C09139=1214.216,61.843,-46.084,-178.985,5.599,148.680
C09140=1214.211,62.093,-46.102,-178.982,5.599,148.680
C09141=1214.206,62.341,-46.118,-178.980,5.600,148.679
C09142=1214.201,62.591,-46.136,-178.978,5.601,148.678
C09143=1214.197,62.841,-46.152,-178.975,5.601,148.678
C09144=1214.192,63.090,-46.169,-178.972,5.602,148.677
C09145=1214.186,63.339,-46.186,-178.970,5.603,148.676
C09146=1214.182,63.589,-46.203,-178.967,5.604,148.676
C09147=1214.177,63.838,-46.220,-178.965,5.604,148.675
C09148=1214.172,64.088,-46.237,-178.962,5.605,148.675
C09149=1214.167,64.337,-46.255,-178.960,5.605,148.674
C09150=1214.162,64.586,-46.271,-178.957,5.606,148.674
C09151=1214.157,64.836,-46.288,-178.954,5.608,148.673
C09152=1214.152,65.085,-46.305,-178.952,5.608,148.672
C09153=1214.147,65.335,-46.322,-178.949,5.609,148.672
C09154=1214.142,65.583,-46.339,-178.947,5.610,148.671
C09155=1214.137,65.833,-46.356,-178.944,5.610,148.670
C09156=1214.133,66.082,-46.373,-178.942,5.611,148.670
C09157=1214.128,66.332,-46.390,-178.939,5.611,148.669
C09158=1214.123,66.582,-46.407,-178.937,5.612,148.669
C09159=1214.118,66.831,-46.425,-178.934,5.613,148.668
C09160=1214.113,67.080,-46.441,-178.932,5.613,148.667
C09161=1214.108,67.329,-46.458,-178.928,5.615,148.667
C09162=1214.103,67.579,-46.475,-178.926,5.616,148.666
C09163=1214.098,67.828,-46.493,-178.924,5.616,148.666
C09164=1214.094,68.078,-46.510,-178.921,5.617,148.665
C09165=1214.088,68.327,-46.527,-178.919,5.618,148.665
C09166=1214.084,68.576,-46.544,-178.916,5.618,148.664
C09167=1214.079,68.825,-46.561,-178.914,5.619,148.663
C09168=1214.074,69.075,-46.579,-178.911,5.619,148.663
C09169=1214.069,69.324,-46.596,-178.909,5.620,148.662
C09170=1214.064,69.574,-46.613,-178.906,5.622,148.662
C09171=1214.060,69.823,-46.630,-178.903,5.622,148.661
C09172=1214.054,70.072,-46.648,-178.900,5.623,148.660
C09173=1214.049,70.322,-46.665,-178.898,5.624,148.660
C09174=1214.044,70.571,-46.681,-178.896,5.624,148.659
C09175=1214.040,70.820,-46.699,-178.893,5.625,148.658
C09176=1214.035,71.070,-46.716,-178.891,5.626,148.658
C09177=1214.030,71.319,-46.733,-178.888,5.626,148.657
C09178=1214.025,71.569,-46.751,-178.885,5.628,148.657
C09179=1214.020,71.818,-46.768,-178.882,5.628,148.656
C09180=1214.016,72.067,-46.786,-178.880,5.629,148.656
C09181=1214.010,72.316,-46.803,-178.878,5.630,148.655
C09182=1214.006,72.565,-46.820,-178.875,5.630,148.654
C09183=1214.000,72.815,-46.838,-178.872,5.631,148.654
C09184=1213.995,73.065,-46.855,-178.870,5.632,148.653
C09185=1213.991,73.314,-46.872,-178.868,5.632,148.653
C09186=1213.986,73.564,-46.889,-178.864,5.634,148.652
C09187=1213.981,73.813,-46.907,-178.862,5.635,148.651
C09188=1213.976,74.062,-46.925,-178.860,5.635,148.651
C09189=1213.971,74.311,-46.942,-178.857,5.636,148.650
C09190=1213.966,74.561,-46.959,-178.854,5.636,148.649
C09191=1213.961,74.810,-46.977,-178.852,5.637,148.649
C09192=1213.957,75.060,-46.994,-178.850,5.638,148.648
C09193=1213.952,75.309,-47.012,-178.846,5.639,148.648
C09194=1213.946,75.557,-47.030,-178.844,5.640,148.647
C09195=1213.941,75.807,-47.047,-178.842,5.641,148.647
C09196=1213.937,76.056,-47.064,-178.839,5.641,148.646
C09197=1213.932,76.306,-47.082,-178.837,5.642,148.646
C09198=1213.927,76.555,-47.099,-178.834,5.643,148.645
C09199=1213.922,76.805,-47.117,-178.831,5.644,148.644
C09200=1213.917,77.054,-47.134,-178.828,5.645,148.644
C09201=1213.913,77.303,-47.152,-178.826,5.646,148.643
C09202=1213.907,77.553,-47.169,-178.824,5.646,148.642
C09203=1213.902,77.802,-47.187,-178.821,5.647,148.642
C09204=1213.898,78.051,-47.205,-178.819,5.648,148.641
C09205=1213.893,78.301,-47.222,-178.816,5.649,148.641
C09206=1213.888,78.550,-47.240,-178.813,5.650,148.640
C09207=1213.883,78.799,-47.258,-178.811,5.651,148.640
C09208=1213.878,79.049,-47.275,-178.808,5.651,148.639
C09209=1213.873,79.298,-47.293,-178.806,5.652,148.638
C09210=1213.868,79.547,-47.311,-178.803,5.653,148.638
C09211=1213.864,79.797,-47.328,-178.801,5.654,148.637
C09212=1213.859,80.046,-47.346,-178.798,5.655,148.637
C09213=1213.854,80.295,-47.364,-178.795,5.655,148.636
C09214=1213.849,80.545,-47.381,-178.793,5.656,148.636
C09215=1213.844,80.794,-47.399,-178.790,5.657,148.635
C09216=1213.839,81.062,-47.418,-178.787,5.658,148.634
C09217=1213.833,81.331,-47.437,-178.784,5.659,148.634
C09218=1213.828,81.599,-47.457,-178.782,5.660,148.633
C09219=1213.823,81.867,-47.476,-178.779,5.661,148.633
C09220=1213.818,82.117,-47.494,-178.776,5.662,148.632
C09221=1213.813,82.366,-47.511,-178.774,5.662,148.631
C09222=1213.808,82.616,-47.529,-178.772,5.663,148.631
C09223=1213.804,82.864,-47.547,-178.769,5.664,148.630
C09224=1213.799,83.114,-47.565,-178.766,5.665,148.629
C09225=1213.794,83.363,-47.583,-178.764,5.666,148.629
C09226=1213.789,83.613,-47.600,-178.761,5.667,148.628
C09227=1213.784,83.862,-47.618,-178.759,5.667,148.628
C09228=1213.779,84.111,-47.636,-178.756,5.668,148.627
C09229=1213.775,84.361,-47.654,-178.754,5.669,148.627
C09230=1213.770,84.610,-47.672,-178.751,5.670,148.626
C09231=1213.765,84.859,-47.690,-178.748,5.671,148.626
C09232=1213.760,85.108,-47.708,-178.746,5.672,148.625
C09233=1213.755,85.358,-47.726,-178.743,5.672,148.624
C09234=1213.750,85.607,-47.743,-178.741,5.673,148.624
C09235=1213.745,85.857,-47.761,-178.738,5.675,148.623
C09236=1213.740,86.106,-47.779,-178.735,5.675,148.623
C09237=1213.735,86.355,-47.797,-178.733,5.676,148.622
C09238=1213.731,86.605,-47.816,-178.730,5.677,148.621
C09239=1213.726,86.854,-47.834,-178.727,5.678,148.621
C09240=1213.721,87.103,-47.852,-178.725,5.679,148.620
C09241=1213.716,87.352,-47.870,-178.723,5.680,148.620
C09242=1213.711,87.601,-47.888,-178.720,5.680,148.619
C09243=1213.706,87.851,-47.905,-178.718,5.681,148.619
C09244=1213.701,88.100,-47.923,-178.715,5.683,148.618
C09245=1213.697,88.350,-47.942,-178.712,5.683,148.617
C09246=1213.692,88.599,-47.960,-178.710,5.684,148.617
C09247=1213.687,88.848,-47.978,-178.707,5.685,148.616
C09248=1213.682,89.098,-47.996,-178.705,5.685,148.616
C09249=1213.677,89.347,-48.014,-178.702,5.687,148.615
C09250=1213.672,89.596,-48.032,-178.699,5.688,148.615
C09251=1213.667,89.846,-48.051,-178.697,5.688,148.614
C09252=1213.662,90.095,-48.069,-178.695,5.689,148.614
C09253=1213.658,90.344,-48.087,-178.691,5.691,148.613
C09254=1213.653,90.593,-48.105,-178.689,5.692,148.612
C09255=1213.648,90.842,-48.123,-178.687,5.692,148.612
C09256=1213.644,91.092,-48.142,-178.684,5.693,148.611
C09257=1213.638,91.341,-48.160,-178.681,5.695,148.611
C09258=1213.633,91.590,-48.178,-178.679,5.695,148.610
C09259=1213.628,91.840,-48.196,-178.676,5.696,148.609
C09260=1213.623,92.089,-48.214,-178.674,5.697,148.609
C09261=1213.619,92.339,-48.232,-178.671,5.698,148.608
C09262=1213.614,92.587,-48.251,-178.668,5.699,148.608
C09263=1213.610,92.836,-48.269,-178.666,5.700,148.607
C09264=1213.604,93.086,-48.288,-178.663,5.700,148.607
C09265=1213.600,93.336,-48.306,-178.661,5.701,148.606
C09266=1213.595,93.585,-48.324,-178.658,5.703,148.606
C09267=1213.590,93.833,-48.343,-178.655,5.703,148.605
C09268=1213.585,94.083,-48.361,-178.653,5.704,148.605
C09269=1213.580,94.333,-48.380,-178.651,5.705,148.604
C09270=1213.575,94.582,-48.398,-178.647,5.706,148.603
C09271=1213.570,94.831,-48.416,-178.645,5.707,148.603
C09272=1213.566,95.080,-48.434,-178.643,5.708,148.602
C09273=1213.561,95.330,-48.453,-178.640,5.709,148.602
C09274=1213.556,95.579,-48.471,-178.637,5.710,148.601
C09275=1213.551,95.828,-48.490,-178.635,5.711,148.600
C09276=1213.546,96.077,-48.508,-178.633,5.711,148.600
C09277=1213.541,96.327,-48.527,-178.629,5.713,148.599
C09278=1213.536,96.576,-48.545,-178.627,5.714,148.599
C09279=1213.532,96.825,-48.564,-178.625,5.714,148.598
C09280=1213.527,97.075,-48.582,-178.622,5.715,148.598
C09281=1213.522,97.324,-48.600,-178.619,5.717,148.597
C09282=1213.517,97.573,-48.619,-178.617,5.717,148.597
C09283=1213.513,97.823,-48.638,-178.615,5.718,148.596
C09284=1213.507,98.072,-48.656,-178.612,5.719,148.596
C09285=1213.502,98.321,-48.675,-178.609,5.720,148.595
C09286=1213.498,98.570,-48.693,-178.607,5.721,148.595
C09287=1213.494,98.819,-48.712,-178.604,5.722,148.594
C09288=1213.488,99.068,-48.730,-178.601,5.724,148.593
C09289=1213.483,99.318,-48.748,-178.599,5.724,148.593
C09290=1213.479,99.567,-48.767,-178.596,5.725,148.592
C09291=1213.473,99.816,-48.786,-178.594,5.726,148.592
C09292=1213.469,100.065,-48.805,-178.591,5.727,148.591
C09293=1213.464,100.315,-48.824,-178.589,5.728,148.591
C09294=1213.459,100.564,-48.842,-178.586,5.729,148.590
C09295=1213.455,100.814,-48.861,-178.583,5.730,148.589
C09296=1213.449,101.062,-48.880,-178.581,5.731,148.589
C09297=1213.445,101.312,-48.898,-178.578,5.732,148.588
C09298=1213.441,101.561,-48.917,-178.576,5.733,148.588
C09299=1213.435,101.810,-48.936,-178.573,5.734,148.587
C09300=1213.430,102.059,-48.954,-178.570,5.735,148.587
C09301=1213.425,102.309,-48.973,-178.568,5.736,148.586
C09302=1213.421,102.558,-48.992,-178.565,5.737,148.586
C09303=1213.416,102.808,-49.011,-178.563,5.738,148.585
C09304=1213.411,103.056,-49.030,-178.560,5.739,148.585
C09305=1213.406,103.306,-49.048,-178.557,5.740,148.584
C09306=1213.401,103.555,-49.067,-178.555,5.741,148.583
C09307=1213.396,103.804,-49.085,-178.552,5.741,148.583
C09308=1213.392,104.054,-49.105,-178.550,5.742,148.582
C09309=1213.387,104.302,-49.124,-178.547,5.744,148.582
C09310=1213.381,104.552,-49.142,-178.545,5.745,148.581
C09311=1213.377,104.801,-49.161,-178.542,5.745,148.581
C09312=1213.372,105.051,-49.180,-178.539,5.747,148.580
C09313=1213.368,105.300,-49.199,-178.537,5.748,148.580
C09314=1213.362,105.549,-49.218,-178.534,5.748,148.579
C09315=1213.358,105.799,-49.236,-178.532,5.750,148.579
C09316=1213.353,106.048,-49.256,-178.529,5.751,148.578
C09317=1213.348,106.296,-49.274,-178.527,5.752,148.578
C09318=1213.343,106.546,-49.293,-178.524,5.753,148.577
C09319=1213.338,106.795,-49.312,-178.522,5.754,148.577
C09320=1213.334,107.064,-49.333,-178.519,5.755,148.576
C09321=1213.328,107.332,-49.353,-178.516,5.756,148.575
C09322=1213.324,107.600,-49.374,-178.513,5.757,148.575
C09323=1213.318,107.869,-49.394,-178.510,5.758,148.574
C09324=1213.313,108.119,-49.413,-178.508,5.759,148.574
C09325=1213.308,108.367,-49.432,-178.505,5.760,148.573
C09326=1213.304,108.617,-49.452,-178.502,5.761,148.573
C09327=1213.298,108.866,-49.470,-178.500,5.762,148.572
C09328=1213.294,109.115,-49.489,-178.497,5.764,148.571
C09329=1213.289,109.364,-49.509,-178.495,5.764,148.571
C09330=1213.285,109.614,-49.528,-178.492,5.765,148.570
C09331=1213.279,109.862,-49.547,-178.489,5.767,148.570
C09332=1213.274,110.113,-49.566,-178.487,5.768,148.569
C09333=1213.270,110.361,-49.585,-178.485,5.768,148.569
C09334=1213.265,110.611,-49.604,-178.482,5.770,148.568
C09335=1213.260,110.859,-49.623,-178.479,5.771,148.568
C09336=1213.256,111.109,-49.643,-178.477,5.772,148.567
C09337=1213.250,111.358,-49.662,-178.474,5.773,148.567
C09338=1213.246,111.608,-49.680,-178.471,5.774,148.566
C09339=1213.241,111.856,-49.700,-178.469,5.775,148.566
C09340=1213.236,112.106,-49.719,-178.466,5.776,148.565
C09341=1213.231,112.355,-49.738,-178.464,5.777,148.565
C09342=1213.226,112.604,-49.758,-178.461,5.778,148.564
C09343=1213.222,112.854,-49.777,-178.459,5.779,148.564
C09344=1213.217,113.102,-49.796,-178.456,5.780,148.563
C09345=1213.212,113.352,-49.816,-178.453,5.782,148.562
C09346=1213.207,113.601,-49.835,-178.451,5.782,148.562
C09347=1213.202,113.850,-49.854,-178.449,5.783,148.561
C09348=1213.198,114.099,-49.873,-178.445,5.785,148.561
C09349=1213.193,114.348,-49.893,-178.443,5.786,148.560
C09350=1213.188,114.598,-49.912,-178.441,5.786,148.560
C09351=1213.184,114.847,-49.931,-178.438,5.788,148.559
C09352=1213.179,115.096,-49.951,-178.435,5.789,148.559
C09353=1213.173,115.345,-49.970,-178.433,5.790,148.558
C09354=1213.169,115.595,-49.990,-178.430,5.791,148.558
C09355=1213.164,115.843,-50.008,-178.428,5.792,148.557
C09356=1213.159,116.093,-50.028,-178.425,5.793,148.557
C09357=1213.155,116.342,-50.048,-178.423,5.794,148.556
C09358=1213.149,116.591,-50.067,-178.420,5.795,148.556
C09359=1213.145,116.841,-50.087,-178.417,5.797,148.555
C09360=1213.141,117.090,-50.106,-178.415,5.797,148.555
C09361=1213.135,117.339,-50.125,-178.412,5.799,148.554
C09362=1213.130,117.588,-50.145,-178.409,5.800,148.553
C09363=1213.125,117.837,-50.164,-178.407,5.801,148.553
C09364=1213.120,118.087,-50.184,-178.404,5.802,148.552
C09365=1213.116,118.336,-50.203,-178.402,5.803,148.552
C09366=1213.111,118.584,-50.223,-178.399,5.804,148.551
C09367=1213.107,118.834,-50.242,-178.397,5.805,148.551
C09368=1213.102,119.083,-50.262,-178.394,5.806,148.550
C09369=1213.097,119.332,-50.281,-178.391,5.808,148.550
C09370=1213.092,119.582,-50.301,-178.389,5.808,148.549
C09371=1213.087,119.831,-50.321,-178.387,5.809,148.549
C09372=1213.083,120.079,-50.340,-178.383,5.811,148.548
C09373=1213.078,120.329,-50.360,-178.381,5.812,148.548
C09374=1213.073,120.579,-50.379,-178.378,5.813,148.547
C09375=1213.068,120.827,-50.399,-178.376,5.814,148.547
C09376=1213.063,121.077,-50.418,-178.373,5.815,148.546
C09377=1213.059,121.326,-50.439,-178.371,5.817,148.546
C09378=1213.054,121.575,-50.458,-178.368,5.817,148.545
C09379=1213.049,121.824,-50.478,-178.365,5.819,148.545
C09380=1213.044,122.074,-50.497,-178.363,5.820,148.544
C09381=1213.039,122.323,-50.518,-178.360,5.821,148.544
C09382=1213.034,122.572,-50.537,-178.358,5.822,148.543
C09383=1213.029,122.821,-50.557,-178.355,5.823,148.543
C09384=1213.026,123.070,-50.576,-178.352,5.824,148.542
C09385=1213.021,123.319,-50.596,-178.350,5.825,148.542
C09386=1213.016,123.568,-50.615,-178.347,5.827,148.541
C09387=1213.011,123.817,-50.636,-178.345,5.828,148.541
C09388=1213.006,124.067,-50.655,-178.342,5.829,148.540
C09389=1213.002,124.316,-50.675,-178.340,5.830,148.540
C09390=1212.997,124.565,-50.695,-178.337,5.831,148.539
C09391=1212.992,124.814,-50.715,-178.334,5.832,148.539
C09392=1212.987,125.064,-50.734,-178.332,5.833,148.538
C09393=1212.983,125.313,-50.755,-178.329,5.835,148.538
C09394=1212.977,125.562,-50.774,-178.327,5.836,148.537
C09395=1212.973,125.811,-50.794,-178.324,5.837,148.537
C09396=1212.968,126.060,-50.814,-178.322,5.838,148.536
C09397=1212.963,126.310,-50.834,-178.319,5.839,148.536
C09398=1212.959,126.559,-50.854,-178.316,5.841,148.535
C09399=1212.953,126.808,-50.874,-178.314,5.841,148.535
C09400=1212.948,127.057,-50.894,-178.311,5.843,148.534
C09401=1212.944,127.306,-50.914,-178.308,5.844,148.533
C09402=1212.939,127.555,-50.934,-178.306,5.845,148.533
C09403=1212.935,127.805,-50.954,-178.304,5.846,148.533
C09404=1212.930,128.053,-50.974,-178.300,5.848,148.532
C09405=1212.925,128.303,-50.994,-178.298,5.849,148.532
C09406=1212.920,128.552,-51.014,-178.296,5.849,148.531
C09407=1212.916,128.801,-51.034,-178.293,5.851,148.531
C09408=1212.911,129.050,-51.054,-178.290,5.852,148.530
C09409=1212.906,129.299,-51.073,-178.288,5.854,148.530
C09410=1212.901,129.548,-51.094,-178.285,5.854,148.529
C09411=1212.896,129.797,-51.115,-178.282,5.856,148.529
C09412=1212.891,130.047,-51.134,-178.280,5.857,148.528
C09413=1212.887,130.296,-51.155,-178.277,5.858,148.528
C09414=1212.882,130.545,-51.174,-178.275,5.859,148.527
C09415=1212.878,130.794,-51.195,-178.272,5.861,148.527
C09416=1212.872,131.043,-51.214,-178.270,5.862,148.526
C09417=1212.867,131.292,-51.235,-178.267,5.863,148.526
C09418=1212.863,131.541,-51.255,-178.264,5.864,148.525
C09419=1212.858,131.791,-51.275,-178.262,5.865,148.525
C09420=1212.854,132.040,-51.295,-178.259,5.867,148.524
C09421=1212.849,132.289,-51.316,-178.257,5.868,148.524
C09422=1212.844,132.539,-51.336,-178.254,5.869,148.523
C09423=1212.839,132.788,-51.356,-178.252,5.870,148.523
C09424=1212.834,133.056,-51.378,-178.249,5.871,148.522
C09425=1212.829,133.325,-51.400,-178.246,5.873,148.522
C09426=1212.823,133.594,-51.422,-178.243,5.874,148.521
C09427=1212.819,133.862,-51.443,-178.241,5.876,148.521
C09428=1212.814,134.111,-51.464,-178.237,5.877,148.520
C09429=1212.809,134.360,-51.484,-178.235,5.878,148.520
C09430=1212.804,134.609,-51.504,-178.232,5.879,148.519
C09431=1212.800,134.858,-51.525,-178.230,5.880,148.519
C09432=1212.795,135.108,-51.546,-178.227,5.882,148.518
C09433=1212.790,135.357,-51.565,-178.225,5.883,148.518
C09434=1212.786,135.606,-51.586,-178.222,5.885,148.517
C09435=1212.781,135.855,-51.606,-178.220,5.885,148.517
C09436=1212.775,136.104,-51.627,-178.217,5.887,148.516
C09437=1212.771,136.353,-51.647,-178.215,5.888,148.516
C09438=1212.767,136.602,-51.667,-178.212,5.889,148.515
C09439=1212.761,136.851,-51.688,-178.209,5.890,148.515
C09440=1212.757,137.100,-51.708,-178.206,5.892,148.514
C09441=1212.752,137.349,-51.728,-178.204,5.893,148.514
C09442=1212.747,137.599,-51.749,-178.201,5.895,148.513
C09443=1212.743,137.848,-51.770,-178.199,5.895,148.513
C09444=1212.738,138.096,-51.790,-178.196,5.897,148.512
C09445=1212.733,138.346,-51.811,-178.194,5.898,148.512
C09446=1212.729,138.595,-51.832,-178.191,5.899,148.511
C09447=1212.724,138.844,-51.851,-178.189,5.900,148.511
C09448=1212.719,139.094,-51.872,-178.186,5.902,148.510
C09449=1212.714,139.342,-51.893,-178.184,5.903,148.510
C09450=1212.709,139.592,-51.913,-178.180,5.904,148.509
C09451=1212.705,139.841,-51.934,-178.178,5.905,148.509
C09452=1212.700,140.090,-51.954,-178.176,5.907,148.509
C09453=1212.695,140.339,-51.975,-178.173,5.908,148.508
C09454=1212.691,140.588,-51.996,-178.170,5.909,148.508
C09455=1212.685,140.837,-52.017,-178.168,5.910,148.507
C09456=1212.681,141.086,-52.037,-178.165,5.912,148.507
C09457=1212.676,141.335,-52.057,-178.163,5.913,148.506
C09458=1212.671,141.584,-52.078,-178.160,5.914,148.506
C09459=1212.667,141.833,-52.099,-178.158,5.915,148.505
C09460=1212.662,142.083,-52.120,-178.155,5.917,148.505
C09461=1212.658,142.332,-52.140,-178.152,5.918,148.504
C09462=1212.653,142.581,-52.161,-178.150,5.919,148.504
C09463=1212.649,142.830,-52.182,-178.147,5.921,148.503
C09464=1212.643,143.079,-52.203,-178.144,5.922,148.503
C09465=1212.639,143.328,-52.224,-178.142,5.924,148.502
C09466=1212.634,143.577,-52.245,-178.140,5.925,148.502
C09467=1212.629,143.826,-52.265,-178.136,5.926,148.501
C09468=1212.624,144.075,-52.286,-178.134,5.927,148.501
C09469=1212.620,144.324,-52.306,-178.132,5.929,148.501
C09470=1212.615,144.574,-52.327,-178.129,5.930,148.500
C09471=1212.610,144.822,-52.348,-178.126,5.931,148.500
C09472=1212.605,145.071,-52.369,-178.124,5.933,148.499
C09473=1212.601,145.321,-52.390,-178.121,5.934,148.499
C09474=1212.596,145.570,-52.411,-178.118,5.936,148.498
C09475=1212.592,145.819,-52.431,-178.116,5.936,148.498
C09476=1212.587,146.068,-52.452,-178.113,5.938,148.497
C09477=1212.582,146.317,-52.474,-178.111,5.939,148.497
C09478=1212.577,146.566,-52.495,-178.108,5.940,148.496
C09479=1212.572,146.815,-52.515,-178.106,5.941,148.496
C09480=1212.568,147.064,-52.536,-178.103,5.943,148.495
C09481=1212.563,147.313,-52.558,-178.100,5.945,148.495
C09482=1212.558,147.563,-52.579,-178.098,5.946,148.494
C09483=1212.554,147.812,-52.599,-178.095,5.947,148.494
C09484=1212.549,148.061,-52.620,-178.093,5.948,148.493
C09485=1212.545,148.309,-52.641,-178.090,5.950,148.493
C09486=1212.539,148.558,-52.662,-178.088,5.951,148.493
C09487=1212.535,148.808,-52.684,-178.085,5.952,148.492
C09488=1212.531,149.057,-52.705,-178.082,5.954,148.492
C09489=1212.525,149.306,-52.726,-178.080,5.955,148.491
C09490=1212.520,149.555,-52.747,-178.077,5.957,148.491
C09491=1212.516,149.804,-52.768,-178.075,5.957,148.490
C09492=1212.511,150.053,-52.789,-178.072,5.959,148.490
C09493=1212.506,150.303,-52.810,-178.069,5.961,148.490
C09494=1212.502,150.551,-52.831,-178.067,5.962,148.489
C09495=1212.497,150.800,-52.852,-178.064,5.963,148.489
C09496=1212.492,151.049,-52.874,-178.062,5.964,148.488
C09497=1212.487,151.298,-52.895,-178.059,5.966,148.488
C09498=1212.484,151.547,-52.916,-178.057,5.967,148.487
C09499=1212.478,151.797,-52.937,-178.054,5.969,148.487
C09500=1212.473,152.046,-52.958,-178.051,5.970,148.486
C09501=1212.469,152.294,-52.979,-178.049,5.971,148.486
C09502=1212.464,152.544,-53.000,-178.046,5.973,148.485
C09503=1212.460,152.793,-53.022,-178.044,5.974,148.485
C09504=1212.454,153.042,-53.043,-178.041,5.975,148.484
C09505=1212.450,153.291,-53.065,-178.038,5.977,148.484
C09506=1212.445,153.540,-53.085,-178.036,5.978,148.484
C09507=1212.441,153.789,-53.107,-178.033,5.980,148.483
C09508=1212.436,154.038,-53.128,-178.030,5.981,148.483
C09509=1212.431,154.287,-53.150,-178.028,5.982,148.482
C09510=1212.426,154.536,-53.170,-178.025,5.984,148.482
C09511=1212.422,154.785,-53.192,-178.023,5.985,148.481
C09512=1212.417,155.034,-53.214,-178.020,5.987,148.481
C09513=1212.412,155.283,-53.235,-178.017,5.988,148.481
C09514=1212.408,155.532,-53.257,-178.015,5.989,148.480
C09515=1212.403,155.782,-53.278,-178.012,5.991,148.480
C09516=1212.398,156.030,-53.299,-178.010,5.992,148.479
C09517=1212.393,156.279,-53.320,-178.007,5.993,148.479
C09518=1212.389,156.529,-53.342,-178.004,5.995,148.478
C09519=1212.384,156.777,-53.364,-178.002,5.996,148.478
C09520=1212.379,157.027,-53.385,-177.999,5.998,148.477
C09521=1212.375,157.276,-53.407,-177.996,5.999,148.477
C09522=1212.370,157.524,-53.428,-177.994,6.000,148.476
C09523=1212.365,157.774,-53.449,-177.992,6.002,148.476
C09524=1212.361,158.023,-53.471,-177.989,6.004,148.476
C09525=1212.356,158.271,-53.493,-177.986,6.005,148.475
C09526=1212.351,158.521,-53.514,-177.984,6.006,148.475
C09527=1212.347,158.770,-53.536,-177.982,6.007,148.474
C09528=1212.342,159.039,-53.560,-177.978,6.009,148.474
C09529=1212.337,159.308,-53.582,-177.976,6.011,148.473
C09530=1212.331,159.577,-53.606,-177.973,6.012,148.473
C09531=1212.327,159.846,-53.629,-177.970,6.014,148.472
C09532=1212.322,160.095,-53.650,-177.967,6.016,148.472
C09533=1212.317,160.344,-53.672,-177.965,6.017,148.472
C09534=1212.313,160.593,-53.694,-177.962,6.018,148.471
C09535=1212.308,160.841,-53.716,-177.959,6.020,148.471
C09536=1212.303,161.091,-53.737,-177.957,6.021,148.470
C09537=1212.298,161.340,-53.759,-177.955,6.023,148.470
C09538=1212.294,161.589,-53.780,-177.952,6.023,148.469
C09539=1212.289,161.838,-53.802,-177.949,6.025,148.469
C09540=1212.284,162.087,-53.824,-177.947,6.027,148.469
C09541=1212.280,162.335,-53.846,-177.945,6.028,148.468
C09542=1212.275,162.585,-53.868,-177.941,6.029,148.468
C09543=1212.270,162.834,-53.889,-177.939,6.031,148.467
C09544=1212.266,163.083,-53.911,-177.937,6.032,148.467
C09545=1212.261,163.332,-53.932,-177.934,6.034,148.466
C09546=1212.256,163.581,-53.954,-177.931,6.036,148.466
C09547=1212.252,163.830,-53.976,-177.929,6.037,148.465
C09548=1212.246,164.079,-53.999,-177.926,6.038,148.465
C09549=1212.242,164.328,-54.021,-177.923,6.040,148.465
C09550=1212.237,164.577,-54.042,-177.920,6.042,148.464
C09551=1212.233,164.826,-54.064,-177.918,6.043,148.464
C09552=1212.228,165.075,-54.086,-177.915,6.044,148.463
C09553=1212.224,165.324,-54.108,-177.913,6.046,148.463
C09554=1212.219,165.573,-54.130,-177.911,6.047,148.463
C09555=1212.214,165.822,-54.152,-177.908,6.049,148.462
C09556=1212.210,166.071,-54.173,-177.905,6.050,148.462
C09557=1212.205,166.319,-54.195,-177.903,6.051,148.461
C09558=1212.200,166.569,-54.217,-177.900,6.053,148.461
C09559=1212.195,166.818,-54.239,-177.897,6.055,148.460
C09560=1212.191,167.067,-54.261,-177.895,6.056,148.460
C09561=1212.186,167.316,-54.283,-177.892,6.058,148.460
C09562=1212.181,167.565,-54.305,-177.890,6.059,148.459
C09563=1212.177,167.814,-54.327,-177.887,6.060,148.459
C09564=1212.172,168.063,-54.349,-177.884,6.062,148.458
C09565=1212.167,168.312,-54.371,-177.882,6.064,148.458
C09566=1212.163,168.561,-54.394,-177.879,6.065,148.458
C09567=1212.158,168.809,-54.416,-177.877,6.066,148.457
C09568=1212.154,169.059,-54.438,-177.874,6.068,148.457
C09569=1212.149,169.307,-54.459,-177.871,6.070,148.456
C09570=1212.144,169.557,-54.482,-177.869,6.071,148.456
C09571=1212.139,169.806,-54.504,-177.866,6.072,148.455
C09572=1212.135,170.054,-54.526,-177.864,6.074,148.455
C09573=1212.131,170.304,-54.549,-177.861,6.076,148.455
C09574=1212.125,170.553,-54.571,-177.858,6.077,148.454
C09575=1212.121,170.802,-54.593,-177.856,6.079,148.454
C09576=1212.116,171.051,-54.615,-177.853,6.080,148.453
C09577=1212.112,171.299,-54.637,-177.851,6.081,148.453
C09578=1212.106,171.548,-54.660,-177.848,6.083,148.453
C09579=1212.102,171.798,-54.682,-177.846,6.085,148.452
C09580=1212.097,172.046,-54.703,-177.842,6.086,148.452
C09581=1212.093,172.295,-54.727,-177.840,6.087,148.451
C09582=1212.088,172.545,-54.749,-177.838,6.089,148.451
C09583=1212.083,172.793,-54.770,-177.835,6.091,148.451
C09584=1212.079,173.043,-54.792,-177.832,6.093,148.450
C09585=1212.074,173.291,-54.815,-177.830,6.094,148.450
C09586=1212.070,173.540,-54.837,-177.827,6.095,148.449
C09587=1212.065,173.790,-54.860,-177.824,6.097,148.449
C09588=1212.060,174.038,-54.883,-177.822,6.099,148.449
C09589=1212.056,174.287,-54.905,-177.820,6.100,148.448
C09590=1212.051,174.535,-54.927,-177.817,6.102,148.448
C09591=1212.046,174.785,-54.950,-177.814,6.103,148.447
C09592=1212.042,175.034,-54.972,-177.811,6.105,148.447
C09593=1212.037,175.283,-54.995,-177.809,6.106,148.446
C09594=1212.032,175.532,-55.017,-177.806,6.108,148.446
C09595=1212.028,175.780,-55.039,-177.804,6.110,148.446
C09596=1212.023,176.030,-55.062,-177.801,6.112,148.445
C09597=1212.018,176.279,-55.084,-177.799,6.113,148.445
C09598=1212.013,176.527,-55.107,-177.796,6.114,148.444
C09599=1212.009,176.777,-55.129,-177.793,6.116,148.444
C09600=1212.005,177.025,-55.152,-177.791,6.118,148.444
C09601=1211.999,177.274,-55.174,-177.789,6.119,148.443
C09602=1211.995,177.523,-55.197,-177.786,6.120,148.443
C09603=1211.990,177.773,-55.219,-177.783,6.122,148.443
C09604=1211.986,178.021,-55.242,-177.781,6.124,148.442
C09605=1211.981,178.270,-55.264,-177.778,6.125,148.442
C09606=1211.977,178.519,-55.287,-177.775,6.127,148.441
C09607=1211.971,178.768,-55.309,-177.773,6.128,148.441
C09608=1211.967,179.017,-55.332,-177.770,6.130,148.441
C09609=1211.963,179.266,-55.356,-177.768,6.131,148.440
C09610=1211.958,179.515,-55.378,-177.765,6.133,148.440
C09611=1211.953,179.763,-55.401,-177.763,6.135,148.439
C09612=1211.949,180.013,-55.423,-177.759,6.136,148.439
C09613=1211.944,180.262,-55.446,-177.757,6.138,148.439
C09614=1211.939,180.510,-55.468,-177.755,6.139,148.438
C09615=1211.934,180.760,-55.491,-177.752,6.141,148.438
C09616=1211.930,181.008,-55.514,-177.749,6.143,148.437
C09617=1211.925,181.258,-55.536,-177.747,6.145,148.437
C09618=1211.921,181.506,-55.559,-177.744,6.146,148.437
C09619=1211.916,181.755,-55.582,-177.742,6.147,148.436
C09620=1211.912,182.004,-55.604,-177.739,6.149,148.436
C09621=1211.907,182.253,-55.628,-177.736,6.151,148.435
C09622=1211.902,182.502,-55.651,-177.734,6.153,148.435
C09623=1211.898,182.750,-55.673,-177.731,6.154,148.435
C09624=1211.893,183.000,-55.696,-177.729,6.155,148.434
C09625=1211.889,183.249,-55.719,-177.726,6.157,148.434
C09626=1211.884,183.497,-55.742,-177.723,6.159,148.434
C09627=1211.879,183.746,-55.765,-177.721,6.161,148.433
C09628=1211.875,183.995,-55.787,-177.718,6.163,148.433
C09629=1211.870,184.245,-55.810,-177.716,6.164,148.432
C09630=1211.866,184.493,-55.833,-177.713,6.165,148.432
C09631=1211.861,184.742,-55.856,-177.710,6.167,148.432
C09632=1211.855,185.011,-55.881,-177.708,6.169,148.431
C09633=1211.851,185.281,-55.906,-177.705,6.171,148.431
C09634=1211.846,185.551,-55.931,-177.702,6.172,148.431
C09635=1211.840,185.820,-55.956,-177.699,6.174,148.430
C09636=1211.836,186.069,-55.979,-177.697,6.176,148.430
C09637=1211.832,186.318,-56.002,-177.694,6.178,148.429
C09638=1211.827,186.567,-56.025,-177.691,6.179,148.429
C09639=1211.823,186.816,-56.047,-177.689,6.180,148.428
C09640=1211.818,187.065,-56.071,-177.686,6.182,148.428
C09641=1211.813,187.314,-56.094,-177.684,6.184,148.428
C09642=1211.808,187.563,-56.117,-177.681,6.186,148.427
C09643=1211.804,187.812,-56.140,-177.679,6.188,148.427
C09644=1211.799,188.061,-56.163,-177.675,6.189,148.427
C09645=1211.795,188.310,-56.187,-177.673,6.190,148.426
C09646=1211.790,188.559,-56.210,-177.671,6.192,148.426
C09647=1211.786,188.807,-56.233,-177.668,6.194,148.425
C09648=1211.781,189.056,-56.256,-177.665,6.196,148.425
C09649=1211.776,189.305,-56.279,-177.663,6.197,148.425
C09650=1211.771,189.554,-56.302,-177.660,6.199,148.424
C09651=1211.767,189.802,-56.325,-177.658,6.200,148.424
C09652=1211.763,190.052,-56.348,-177.655,6.202,148.424
C09653=1211.758,190.301,-56.372,-177.653,6.204,148.423
C09654=1211.753,190.550,-56.395,-177.650,6.206,148.423
C09655=1211.748,190.799,-56.419,-177.647,6.208,148.423
C09656=1211.744,191.047,-56.441,-177.645,6.209,148.422
C09657=1211.740,191.296,-56.465,-177.642,6.211,148.422
C09658=1211.734,191.545,-56.488,-177.640,6.212,148.422
C09659=1211.730,191.794,-56.511,-177.637,6.214,148.421
C09660=1211.725,192.042,-56.535,-177.634,6.216,148.421
C09661=1211.721,192.291,-56.558,-177.631,6.217,148.420
C09662=1211.716,192.540,-56.582,-177.629,6.219,148.420
C09663=1211.711,192.789,-56.605,-177.626,6.221,148.420
C09664=1211.707,193.038,-56.628,-177.624,6.223,148.419
C09665=1211.703,193.287,-56.651,-177.621,6.224,148.419
C09666=1211.698,193.536,-56.675,-177.619,6.226,148.418
C09667=1211.694,193.784,-56.699,-177.616,6.227,148.418
C09668=1211.689,194.033,-56.722,-177.613,6.229,148.418
C09669=1211.684,194.283,-56.745,-177.611,6.231,148.417
C09670=1211.679,194.532,-56.769,-177.608,6.233,148.417
C09671=1211.675,194.781,-56.792,-177.606,6.235,148.417
C09672=1211.670,195.029,-56.816,-177.603,6.237,148.416
C09673=1211.666,195.278,-56.840,-177.601,6.238,148.416
C09674=1211.661,195.527,-56.863,-177.598,6.239,148.416
C09675=1211.656,195.776,-56.886,-177.596,6.241,148.415
C09676=1211.652,196.024,-56.910,-177.593,6.243,148.415
C09677=1211.647,196.274,-56.934,-177.590,6.245,148.415
C09678=1211.642,196.523,-56.957,-177.588,6.247,148.414
C09679=1211.638,196.771,-56.981,-177.585,6.249,148.414
C09680=1211.633,197.020,-57.005,-177.582,6.250,148.414
C09681=1211.629,197.269,-57.028,-177.580,6.252,148.413
C09682=1211.624,197.517,-57.052,-177.578,6.253,148.413
C09683=1211.620,197.766,-57.075,-177.575,6.255,148.413
C09684=1211.615,198.016,-57.099,-177.572,6.257,148.412
C09685=1211.610,198.264,-57.123,-177.570,6.259,148.412
C09686=1211.606,198.513,-57.146,-177.567,6.261,148.412
C09687=1211.601,198.761,-57.170,-177.564,6.262,148.411
C09688=1211.597,199.010,-57.194,-177.562,6.264,148.411
C09689=1211.592,199.259,-57.217,-177.559,6.266,148.410
C09690=1211.588,199.508,-57.241,-177.556,6.268,148.410
C09691=1211.583,199.757,-57.264,-177.554,6.270,148.410
C09692=1211.578,200.005,-57.288,-177.551,6.272,148.409
C09693=1211.574,200.254,-57.312,-177.549,6.273,148.409
C09694=1211.569,200.503,-57.336,-177.546,6.274,148.409
C09695=1211.565,200.752,-57.359,-177.544,6.276,148.408
C09696=1211.560,201.001,-57.384,-177.541,6.278,148.408
C09697=1211.555,201.250,-57.408,-177.538,6.280,148.408
C09698=1211.551,201.499,-57.432,-177.536,6.282,148.407
C09699=1211.546,201.748,-57.455,-177.533,6.284,148.407
C09700=1211.542,201.996,-57.479,-177.530,6.285,148.407
C09701=1211.537,202.245,-57.502,-177.528,6.287,148.406
C09702=1211.533,202.494,-57.527,-177.525,6.289,148.406
C09703=1211.527,202.743,-57.551,-177.523,6.291,148.406
C09704=1211.523,202.991,-57.575,-177.520,6.293,148.405
C09705=1211.519,203.240,-57.599,-177.517,6.295,148.405
C09706=1211.515,203.489,-57.622,-177.515,6.296,148.405
C09707=1211.510,203.738,-57.646,-177.513,6.297,148.404
C09708=1211.506,203.986,-57.671,-177.510,6.299,148.404
C09709=1211.500,204.236,-57.694,-177.507,6.301,148.404
C09710=1211.496,204.484,-57.719,-177.505,6.303,148.403
C09711=1211.491,204.733,-57.742,-177.502,6.305,148.403
C09712=1211.487,204.982,-57.766,-177.499,6.307,148.403
C09713=1211.482,205.231,-57.791,-177.497,6.308,148.402
C09714=1211.478,205.479,-57.815,-177.494,6.310,148.402
C09715=1211.473,205.728,-57.838,-177.491,6.312,148.402
C09716=1211.469,205.977,-57.863,-177.489,6.314,148.401
C09717=1211.464,206.226,-57.888,-177.486,6.316,148.401
C09718=1211.460,206.475,-57.911,-177.483,6.318,148.401
C09719=1211.455,206.724,-57.935,-177.481,6.319,148.400
C09720=1211.451,206.972,-57.959,-177.478,6.321,148.400
C09721=1211.446,207.221,-57.984,-177.475,6.323,148.400
C09722=1211.441,207.470,-58.007,-177.473,6.325,148.399
C09723=1211.437,207.719,-58.032,-177.471,6.327,148.399
C09724=1211.432,207.968,-58.056,-177.468,6.329,148.399
C09725=1211.428,208.216,-58.080,-177.465,6.331,148.398
C09726=1211.423,208.464,-58.104,-177.463,6.333,148.398
C09727=1211.419,208.714,-58.129,-177.460,6.334,148.398
C09728=1211.414,208.963,-58.153,-177.458,6.335,148.397
C09729=1211.410,209.211,-58.177,-177.455,6.337,148.397
C09730=1211.404,209.460,-58.201,-177.453,6.339,148.397
C09731=1211.401,209.709,-58.226,-177.450,6.341,148.396
C09732=1211.396,209.958,-58.251,-177.447,6.343,148.396
C09733=1211.391,210.206,-58.275,-177.445,6.345,148.396
C09734=1211.387,210.455,-58.299,-177.442,6.346,148.395
C09735=1211.382,210.704,-58.324,-177.440,6.348,148.395
C09736=1211.377,210.975,-58.350,-177.436,6.351,148.395
C09737=1211.372,211.245,-58.376,-177.434,6.353,148.394
C09738=1211.367,211.515,-58.403,-177.431,6.355,148.394
C09739=1211.362,211.785,-58.429,-177.428,6.356,148.394
C09740=1211.358,212.034,-58.454,-177.426,6.358,148.393
C09741=1211.353,212.283,-58.478,-177.423,6.360,148.393
C09742=1211.349,212.531,-58.503,-177.421,6.362,148.393
C09743=1211.344,212.781,-58.528,-177.418,6.364,148.392
C09744=1211.340,213.029,-58.552,-177.415,6.366,148.392
C09745=1211.335,213.278,-58.576,-177.413,6.368,148.392
C09746=1211.331,213.527,-58.601,-177.410,6.370,148.392
C09747=1211.326,213.776,-58.625,-177.408,6.372,148.391
C09748=1211.321,214.024,-58.649,-177.405,6.373,148.391
C09749=1211.317,214.274,-58.675,-177.403,6.375,148.391
C09750=1211.312,214.522,-58.699,-177.400,6.377,148.390
C09751=1211.307,214.771,-58.723,-177.397,6.379,148.390
C09752=1211.304,215.020,-58.748,-177.395,6.381,148.390
C09753=1211.298,215.269,-58.772,-177.392,6.383,148.389
C09754=1211.294,215.516,-58.797,-177.389,6.384,148.389
C09755=1211.290,215.766,-58.822,-177.387,6.386,148.389
C09756=1211.285,216.014,-58.846,-177.385,6.388,148.388
C09757=1211.280,216.263,-58.871,-177.381,6.391,148.388
C09758=1211.276,216.512,-58.896,-177.379,6.393,148.388
C09759=1211.271,216.761,-58.920,-177.376,6.395,148.387
C09760=1211.266,217.009,-58.945,-177.373,6.397,148.387
C09761=1211.263,217.258,-58.970,-177.371,6.398,148.387
C09762=1211.258,217.507,-58.995,-177.368,6.400,148.387
C09763=1211.253,217.756,-59.020,-177.365,6.402,148.386
C09764=1211.249,218.004,-59.044,-177.363,6.404,148.386
C09765=1211.244,218.253,-59.069,-177.361,6.406,148.386
C09766=1211.240,218.502,-59.093,-177.358,6.408,148.385
C09767=1211.235,218.750,-59.118,-177.355,6.410,148.385
C09768=1211.231,218.999,-59.144,-177.353,6.412,148.385
C09769=1211.226,219.248,-59.168,-177.350,6.414,148.384
C09770=1211.222,219.497,-59.193,-177.348,6.415,148.384
C09771=1211.217,219.745,-59.218,-177.345,6.417,148.384
C09772=1211.213,219.994,-59.242,-177.343,6.419,148.384
C09773=1211.208,220.243,-59.267,-177.340,6.421,148.383
C09774=1211.203,220.491,-59.293,-177.337,6.423,148.383
C09775=1211.199,220.740,-59.317,-177.335,6.425,148.383
C09776=1211.194,220.989,-59.342,-177.332,6.427,148.382
C09777=1211.190,221.238,-59.368,-177.330,6.429,148.382
C09778=1211.185,221.487,-59.392,-177.327,6.430,148.382
C09779=1211.181,221.735,-59.418,-177.325,6.433,148.382
C09780=1211.176,221.984,-59.442,-177.322,6.434,148.381
C09781=1211.172,222.233,-59.468,-177.319,6.436,148.381
C09782=1211.167,222.481,-59.493,-177.317,6.438,148.381
C09783=1211.163,222.730,-59.517,-177.314,6.440,148.380
C09784=1211.158,222.978,-59.542,-177.312,6.442,148.380
C09785=1211.154,223.228,-59.568,-177.309,6.445,148.380
C09786=1211.149,223.476,-59.593,-177.306,6.447,148.380
C09787=1211.145,223.725,-59.617,-177.304,6.449,148.379
C09788=1211.140,223.973,-59.643,-177.301,6.450,148.379
C09789=1211.136,224.223,-59.668,-177.298,6.452,148.379
C09790=1211.131,224.471,-59.693,-177.296,6.454,148.378
C09791=1211.127,224.720,-59.719,-177.294,6.456,148.378
C09792=1211.122,224.968,-59.743,-177.291,6.458,148.378
C09793=1211.118,225.217,-59.769,-177.288,6.460,148.377
C09794=1211.113,225.466,-59.793,-177.286,6.462,148.377
C09795=1211.109,225.714,-59.819,-177.283,6.464,148.377
C09796=1211.104,225.963,-59.844,-177.281,6.466,148.377
C09797=1211.099,226.212,-59.870,-177.278,6.468,148.376
C09798=1211.095,226.460,-59.895,-177.276,6.469,148.376
C09799=1211.091,226.709,-59.919,-177.273,6.471,148.376
C09800=1211.086,226.957,-59.945,-177.270,6.473,148.375
C09801=1211.082,227.206,-59.971,-177.268,6.475,148.375
C09802=1211.077,227.455,-59.996,-177.265,6.478,148.375
C09803=1211.072,227.703,-60.021,-177.262,6.480,148.375
C09804=1211.068,227.952,-60.047,-177.260,6.482,148.374
C09805=1211.063,228.201,-60.071,-177.257,6.484,148.374
C09806=1211.059,228.450,-60.097,-177.255,6.486,148.374
C09807=1211.055,228.699,-60.123,-177.252,6.488,148.374
C09808=1211.050,228.947,-60.148,-177.250,6.489,148.373
C09809=1211.045,229.196,-60.173,-177.247,6.491,148.373
C09810=1211.040,229.444,-60.199,-177.244,6.493,148.373
C09811=1211.036,229.693,-60.224,-177.242,6.495,148.373
C09812=1211.032,229.942,-60.250,-177.240,6.497,148.372
C09813=1211.028,230.190,-60.274,-177.237,6.499,148.372
C09814=1211.023,230.439,-60.300,-177.234,6.502,148.372
C09815=1211.018,230.687,-60.325,-177.232,6.504,148.371
C09816=1211.014,230.936,-60.351,-177.229,6.506,148.371
C09817=1211.010,231.185,-60.377,-177.226,6.508,148.371
C09818=1211.005,231.433,-60.402,-177.224,6.509,148.371
C09819=1211.000,231.683,-60.428,-177.222,6.512,148.370
C09820=1210.996,231.931,-60.454,-177.219,6.513,148.370
C09821=1210.991,232.180,-60.479,-177.216,6.515,148.370
C09822=1210.987,232.428,-60.505,-177.214,6.517,148.369
C09823=1210.982,232.677,-60.531,-177.212,6.519,148.369
C09824=1210.978,232.925,-60.556,-177.209,6.521,148.369
C09825=1210.973,233.174,-60.582,-177.206,6.524,148.369
C09826=1210.969,233.423,-60.607,-177.203,6.526,148.368
C09827=1210.964,233.671,-60.633,-177.201,6.528,148.368
C09828=1210.960,233.920,-60.659,-177.198,6.530,148.368
C09829=1210.956,234.169,-60.684,-177.196,6.532,148.368
C09830=1210.951,234.417,-60.710,-177.193,6.533,148.367
C09831=1210.947,234.665,-60.735,-177.191,6.536,148.367
C09832=1210.942,234.915,-60.762,-177.188,6.537,148.367
C09833=1210.938,235.163,-60.788,-177.186,6.539,148.367
C09834=1210.933,235.412,-60.813,-177.182,6.542,148.366
C09835=1210.929,235.660,-60.839,-177.180,6.544,148.366
C09836=1210.924,235.909,-60.864,-177.178,6.546,148.366
C09837=1210.920,236.158,-60.890,-177.175,6.548,148.366
C09838=1210.915,236.406,-60.916,-177.172,6.550,148.365
C09839=1210.910,236.655,-60.942,-177.170,6.552,148.365
C09840=1210.906,236.927,-60.970,-177.167,6.555,148.365
C09841=1210.901,237.198,-60.998,-177.164,6.556,148.365
C09842=1210.896,237.470,-61.026,-177.162,6.558,148.364
C09843=1210.892,237.741,-61.055,-177.159,6.561,148.364
C09844=1210.887,237.989,-61.081,-177.157,6.563,148.364
C09845=1210.883,238.238,-61.106,-177.154,6.565,148.364
C09846=1210.878,238.487,-61.133,-177.151,6.567,148.363
C09847=1210.873,238.736,-61.158,-177.149,6.569,148.363
C09848=1210.869,238.984,-61.184,-177.147,6.571,148.363
C09849=1210.865,239.232,-61.210,-177.143,6.574,148.363
C09850=1210.860,239.481,-61.237,-177.141,6.575,148.362
C09851=1210.855,239.730,-61.262,-177.139,6.578,148.362
C09852=1210.851,239.979,-61.288,-177.136,6.579,148.362
C09853=1210.846,240.226,-61.315,-177.133,6.581,148.362
C09854=1210.842,240.475,-61.341,-177.131,6.584,148.361
C09855=1210.838,240.724,-61.366,-177.129,6.585,148.361
C09856=1210.833,240.973,-61.392,-177.125,6.588,148.361
C09857=1210.829,241.221,-61.419,-177.123,6.590,148.361
C09858=1210.824,241.469,-61.444,-177.121,6.592,148.360
C09859=1210.820,241.718,-61.470,-177.118,6.594,148.360
C09860=1210.815,241.967,-61.497,-177.116,6.596,148.360
C09861=1210.811,242.216,-61.523,-177.113,6.598,148.360
C09862=1210.806,242.464,-61.549,-177.111,6.600,148.359
C09863=1210.802,242.713,-61.576,-177.108,6.603,148.359
C09864=1210.798,242.962,-61.602,-177.105,6.605,148.359
C09865=1210.792,243.210,-61.628,-177.103,6.607,148.359
C09866=1210.788,243.458,-61.654,-177.100,6.609,148.359
C09867=1210.784,243.707,-61.680,-177.098,6.611,148.358
C09868=1210.779,243.956,-61.707,-177.095,6.612,148.358
C09869=1210.775,244.204,-61.733,-177.092,6.615,148.358
C09870=1210.770,244.453,-61.760,-177.090,6.617,148.358
C09871=1210.766,244.702,-61.785,-177.087,6.619,148.357
C09872=1210.762,244.950,-61.811,-177.085,6.621,148.357
C09873=1210.757,245.198,-61.838,-177.082,6.623,148.357
C09874=1210.752,245.447,-61.864,-177.080,6.625,148.357
C09875=1210.748,245.696,-61.891,-177.077,6.628,148.356
C09876=1210.744,245.944,-61.916,-177.075,6.630,148.356
C09877=1210.739,246.193,-61.943,-177.072,6.632,148.356
C09878=1210.735,246.441,-61.970,-177.070,6.634,148.356
C09879=1210.730,246.690,-61.996,-177.067,6.636,148.355
C09880=1210.726,246.938,-62.023,-177.064,6.639,148.355
C09881=1210.721,247.187,-62.049,-177.062,6.641,148.355
C09882=1210.717,247.436,-62.076,-177.059,6.643,148.355
C09883=1210.712,247.685,-62.102,-177.057,6.645,148.355
C09884=1210.708,247.933,-62.128,-177.054,6.647,148.354
C09885=1210.704,248.181,-62.155,-177.051,6.649,148.354
C09886=1210.699,248.430,-62.181,-177.049,6.651,148.354
C09887=1210.695,248.679,-62.208,-177.046,6.653,148.354
C09888=1210.691,248.928,-62.234,-177.044,6.656,148.354
C09889=1210.686,249.176,-62.261,-177.042,6.657,148.353
C09890=1210.681,249.424,-62.287,-177.039,6.660,148.353
C09891=1210.677,249.672,-62.314,-177.036,6.662,148.353
C09892=1210.672,249.921,-62.340,-177.034,6.664,148.353
C09893=1210.668,250.169,-62.367,-177.032,6.666,148.353
C09894=1210.663,250.418,-62.394,-177.029,6.668,148.352
C09895=1210.659,250.667,-62.420,-177.026,6.671,148.352
C09896=1210.654,250.915,-62.447,-177.024,6.673,148.352
C09897=1210.650,251.163,-62.473,-177.021,6.675,148.352
C09898=1210.646,251.412,-62.500,-177.019,6.677,148.351
C09899=1210.641,251.662,-62.527,-177.016,6.679,148.351
C09900=1210.637,251.910,-62.554,-177.013,6.682,148.351
C09901=1210.633,252.158,-62.581,-177.011,6.684,148.351
C09902=1210.628,252.407,-62.608,-177.008,6.686,148.350
C09903=1210.624,252.655,-62.634,-177.006,6.688,148.350
C09904=1210.619,252.904,-62.661,-177.004,6.690,148.350
C09905=1210.615,253.153,-62.688,-177.000,6.692,148.350
C09906=1210.611,253.401,-62.714,-176.998,6.695,148.350
C09907=1210.606,253.649,-62.741,-176.996,6.696,148.349
C09908=1210.601,253.898,-62.768,-176.994,6.699,148.349
C09909=1210.597,254.146,-62.795,-176.990,6.701,148.349
C09910=1210.593,254.394,-62.822,-176.988,6.704,148.349
C09911=1210.588,254.643,-62.849,-176.986,6.705,148.349
C09912=1210.583,254.891,-62.876,-176.983,6.707,148.348
C09913=1210.579,255.140,-62.902,-176.980,6.710,148.348
C09914=1210.575,255.389,-62.929,-176.978,6.712,148.348
C09915=1210.570,255.637,-62.956,-176.976,6.714,148.348
C09916=1210.566,255.886,-62.983,-176.973,6.716,148.348
C09917=1210.562,256.135,-63.010,-176.970,6.719,148.348
C09918=1210.557,256.383,-63.037,-176.968,6.721,148.347
C09919=1210.553,256.632,-63.064,-176.965,6.723,148.347
C09920=1210.548,256.880,-63.091,-176.963,6.725,148.347
C09921=1210.544,257.128,-63.117,-176.960,6.728,148.347
C09922=1210.539,257.377,-63.144,-176.957,6.730,148.347
C09923=1210.535,257.625,-63.172,-176.955,6.732,148.346
C09924=1210.531,257.874,-63.200,-176.953,6.734,148.346
C09925=1210.526,258.122,-63.227,-176.950,6.737,148.346
C09926=1210.522,258.371,-63.254,-176.947,6.739,148.346
C09927=1210.518,258.619,-63.280,-176.945,6.741,148.345
C09928=1210.513,258.868,-63.307,-176.943,6.743,148.345
C09929=1210.508,259.116,-63.334,-176.939,6.746,148.345
C09930=1210.504,259.365,-63.361,-176.937,6.748,148.345
C09931=1210.500,259.614,-63.389,-176.935,6.750,148.345
C09932=1210.495,259.862,-63.417,-176.933,6.752,148.345
C09933=1210.491,260.110,-63.444,-176.929,6.755,148.344
C09934=1210.486,260.359,-63.471,-176.927,6.757,148.344
C09935=1210.482,260.607,-63.497,-176.925,6.759,148.344
C09936=1210.478,260.856,-63.525,-176.922,6.762,148.344
C09937=1210.473,261.104,-63.552,-176.919,6.764,148.344
C09938=1210.469,261.352,-63.579,-176.917,6.766,148.344
C09939=1210.464,261.601,-63.606,-176.915,6.768,148.343
C09940=1210.460,261.849,-63.634,-176.912,6.771,148.343
C09941=1210.456,262.099,-63.661,-176.909,6.772,148.343
C09942=1210.451,262.346,-63.689,-176.907,6.775,148.343
C09943=1210.447,262.595,-63.716,-176.904,6.777,148.343
C09944=1210.442,262.867,-63.745,-176.902,6.780,148.343
C09945=1210.437,263.140,-63.776,-176.899,6.782,148.342
C09946=1210.432,263.413,-63.806,-176.896,6.784,148.342
C09947=1210.428,263.685,-63.836,-176.893,6.787,148.342
C09948=1210.423,263.934,-63.863,-176.891,6.789,148.342
C09949=1210.418,264.182,-63.890,-176.888,6.792,148.342
C09950=1210.415,264.431,-63.918,-176.885,6.794,148.341
C09951=1210.410,264.680,-63.946,-176.883,6.796,148.341
C09952=1210.405,264.928,-63.973,-176.880,6.799,148.341
C09953=1210.401,265.176,-64.000,-176.878,6.801,148.341
C09954=1210.397,265.425,-64.028,-176.875,6.803,148.341
C09955=1210.393,265.673,-64.056,-176.873,6.805,148.340
C09956=1210.388,265.921,-64.083,-176.870,6.808,148.340
C09957=1210.383,266.170,-64.111,-176.868,6.810,148.340
C09958=1210.379,266.419,-64.138,-176.866,6.812,148.340
C09959=1210.374,266.667,-64.165,-176.863,6.815,148.340
C09960=1210.370,266.915,-64.193,-176.860,6.817,148.340
C09961=1210.366,267.164,-64.221,-176.858,6.819,148.339
C09962=1210.361,267.412,-64.248,-176.855,6.822,148.339
C09963=1210.357,267.660,-64.276,-176.853,6.824,148.339
C09964=1210.353,267.909,-64.304,-176.850,6.826,148.339
C09965=1210.349,268.157,-64.331,-176.847,6.829,148.339
C09966=1210.343,268.406,-64.359,-176.845,6.831,148.339
C09967=1210.340,268.655,-64.387,-176.843,6.833,148.339
C09968=1210.335,268.903,-64.414,-176.840,6.836,148.338
C09969=1210.330,269.151,-64.442,-176.838,6.838,148.338
C09970=1210.327,269.400,-64.470,-176.835,6.840,148.338
C09971=1210.321,269.648,-64.498,-176.832,6.843,148.338
C09972=1210.317,269.896,-64.526,-176.830,6.845,148.338
C09973=1210.313,270.145,-64.553,-176.828,6.847,148.338
C09974=1210.309,270.393,-64.581,-176.825,6.850,148.337
C09975=1210.305,270.642,-64.609,-176.822,6.852,148.337
C09976=1210.299,270.891,-64.637,-176.820,6.854,148.337
C09977=1210.295,271.139,-64.664,-176.817,6.857,148.337
C09978=1210.291,271.387,-64.693,-176.815,6.859,148.337
C09979=1210.287,271.635,-64.720,-176.813,6.861,148.337
C09980=1210.282,271.884,-64.748,-176.810,6.864,148.336
C09981=1210.278,272.132,-64.776,-176.807,6.866,148.336
C09982=1210.274,272.380,-64.804,-176.804,6.869,148.336
C09983=1210.269,272.629,-64.831,-176.802,6.871,148.336
C09984=1210.264,272.878,-64.860,-176.800,6.873,148.336
C09985=1210.261,273.126,-64.888,-176.797,6.876,148.336
C09986=1210.256,273.374,-64.916,-176.795,6.878,148.336
C09987=1210.251,273.622,-64.944,-176.792,6.880,148.335
C09988=1210.247,273.872,-64.971,-176.789,6.883,148.335
C09989=1210.243,274.119,-64.999,-176.787,6.885,148.335
C09990=1210.239,274.368,-65.027,-176.785,6.887,148.335
C09991=1210.234,274.616,-65.056,-176.782,6.890,148.335
C09992=1210.230,274.865,-65.084,-176.780,6.892,148.335
C09993=1210.225,275.113,-65.112,-176.777,6.895,148.335
C09994=1210.221,275.361,-65.140,-176.775,6.897,148.335
C09995=1210.217,275.609,-65.168,-176.772,6.899,148.334
C09996=1210.212,275.859,-65.196,-176.769,6.902,148.334
//INST
///DATE 2021/06/25 14:27
///ATTR SC,RW,RJ
////FRAME ROBOT
///GROUP1 RB1
NOP
MOVL C00000 V=800.0 PL=0
MOVL C00001 V=800.0 PL=0
MOVL C00002 V=800.0 PL=0
MOVL C00003 V=800.0 PL=0
MOVL C00004 V=800.0 PL=0
MOVL C00005 V=800.0 PL=0
MOVL C00006 V=800.0 PL=0
MOVL C00007 V=800.0 PL=0
MOVL C00008 V=800.0 PL=0
MOVL C00009 V=800.0 PL=0
MOVL C00010 V=800.0 PL=0
MOVL C00011 V=800.0 PL=0
MOVL C00012 V=800.0 PL=0
MOVL C00013 V=800.0 PL=0
MOVL C00014 V=800.0 PL=0
MOVL C00015 V=800.0 PL=0
MOVL C00016 V=800.0 PL=0
MOVL C00017 V=800.0 PL=0
MOVL C00018 V=800.0 PL=0
MOVL C00019 V=800.0 PL=0
MOVL C00020 V=800.0 PL=0
MOVL C00021 V=800.0 PL=0
MOVL C00022 V=800.0 PL=0
MOVL C00023 V=800.0 PL=0
MOVL C00024 V=800.0 PL=0
MOVL C00025 V=800.0 PL=0
MOVL C00026 V=800.0 PL=0
MOVL C00027 V=800.0 PL=0
MOVL C00028 V=800.0 PL=0
MOVL C00029 V=800.0 PL=0
MOVL C00030 V=800.0 PL=0
MOVL C00031 V=800.0 PL=0
MOVL C00032 V=800.0 PL=0
MOVL C00033 V=800.0 PL=0
MOVL C00034 V=800.0 PL=0
MOVL C00035 V=800.0 PL=0
MOVL C00036 V=800.0 PL=0
MOVL C00037 V=800.0 PL=0
MOVL C00038 V=800.0 PL=0
MOVL C00039 V=800.0 PL=0
MOVL C00040 V=800.0 PL=0
MOVL C00041 V=800.0 PL=0
MOVL C00042 V=800.0 PL=0
MOVL C00043 V=800.0 PL=0
MOVL C00044 V=800.0 PL=0
MOVL C00045 V=800.0 PL=0
MOVL C00046 V=800.0 PL=0
MOVL C00047 V=800.0 PL=0
MOVL C00048 V=800.0 PL=0
MOVL C00049 V=800.0 PL=0
MOVL C00050 V=800.0 PL=0
MOVL C00051 V=800.0 PL=0
MOVL C00052 V=800.0 PL=0
MOVL C00053 V=800.0 PL=0
MOVL C00054 V=800.0 PL=0
MOVL C00055 V=800.0 PL=0
MOVL C00056 V=800.0 PL=0
MOVL C00057 V=800.0 PL=0
MOVL C00058 V=800.0 PL=0
MOVL C00059 V=800.0 PL=0
MOVL C00060 V=800.0 PL=0
MOVL C00061 V=800.0 PL=0
MOVL C00062 V=800.0 PL=0
MOVL C00063 V=800.0 PL=0
MOVL C00064 V=800.0 PL=0
MOVL C00065 V=800.0 PL=0
MOVL C00066 V=800.0 PL=0
MOVL C00067 V=800.0 PL=0
MOVL C00068 V=800.0 PL=0
MOVL C00069 V=800.0 PL=0
MOVL C00070 V=800.0 PL=0
MOVL C00071 V=800.0 PL=0
MOVL C00072 V=800.0 PL=0
MOVL C00073 V=800.0 PL=0
MOVL C00074 V=800.0 PL=0
MOVL C00075 V=800.0 PL=0
MOVL C00076 V=800.0 PL=0
MOVL C00077 V=800.0 PL=0
MOVL C00078 V=800.0 PL=0
MOVL C00079 V=800.0 PL=0
MOVL C00080 V=800.0 PL=0
MOVL C00081 V=800.0 PL=0
MOVL C00082 V=800.0 PL=0
MOVL C00083 V=800.0 PL=0
MOVL C00084 V=800.0 PL=0
MOVL C00085 V=800.0 PL=0
MOVL C00086 V=800.0 PL=0
MOVL C00087 V=800.0 PL=0
MOVL C00088 V=800.0 PL=0
MOVL C00089 V=800.0 PL=0
MOVL C00090 V=800.0 PL=0
MOVL C00091 V=800.0 PL=0
MOVL C00092 V=800.0 PL=0
MOVL C00093 V=800.0 PL=0
MOVL C00094 V=800.0 PL=0
MOVL C00095 V=800.0 PL=0
MOVL C00096 V=800.0 PL=0
MOVL C00097 V=800.0 PL=0
MOVL C00098 V=800.0 PL=0
MOVL C00099 V=800.0 PL=0
MOVL C00100 V=800.0 PL=0
MOVL C00101 V=800.0 PL=0
MOVL C00102 V=800.0 PL=0
MOVL C00103 V=800.0 PL=0
MOVL C00104 V=800.0 PL=0
MOVL C00105 V=800.0 PL=0
MOVL C00106 V=800.0 PL=0
MOVL C00107 V=800.0 PL=0
MOVL C00108 V=800.0 PL=0
MOVL C00109 V=800.0 PL=0
MOVL C00110 V=800.0 PL=0
MOVL C00111 V=800.0 PL=0
MOVL C00112 V=800.0 PL=0
MOVL C00113 V=800.0 PL=0
MOVL C00114 V=800.0 PL=0
MOVL C00115 V=800.0 PL=0
MOVL C00116 V=800.0 PL=0
MOVL C00117 V=800.0 PL=0
MOVL C00118 V=800.0 PL=0
MOVL C00119 V=800.0 PL=0
MOVL C00120 V=800.0 PL=0
MOVL C00121 V=800.0 PL=0
MOVL C00122 V=800.0 PL=0
MOVL C00123 V=800.0 PL=0
MOVL C00124 V=800.0 PL=0
MOVL C00125 V=800.0 PL=0
MOVL C00126 V=800.0 PL=0
MOVL C00127 V=800.0 PL=0
MOVL C00128 V=800.0 PL=0
MOVL C00129 V=800.0 PL=0
MOVL C00130 V=800.0 PL=0
MOVL C00131 V=800.0 PL=0
MOVL C00132 V=800.0 PL=0
MOVL C00133 V=800.0 PL=0
MOVL C00134 V=800.0 PL=0
MOVL C00135 V=800.0 PL=0
MOVL C00136 V=800.0 PL=0
MOVL C00137 V=800.0 PL=0
MOVL C00138 V=800.0 PL=0
MOVL C00139 V=800.0 PL=0
MOVL C00140 V=800.0 PL=0
MOVL C00141 V=800.0 PL=0
MOVL C00142 V=800.0 PL=0
MOVL C00143 V=800.0 PL=0
MOVL C00144 V=800.0 PL=0
MOVL C00145 V=800.0 PL=0
MOVL C00146 V=800.0 PL=0
MOVL C00147 V=800.0 PL=0
MOVL C00148 V=800.0 PL=0
MOVL C00149 V=800.0 PL=0
MOVL C00150 V=800.0 PL=0
MOVL C00151 V=800.0 PL=0
MOVL C00152 V=800.0 PL=0
MOVL C00153 V=800.0 PL=0
MOVL C00154 V=800.0 PL=0
MOVL C00155 V=800.0 PL=0
MOVL C00156 V=800.0 PL=0
MOVL C00157 V=800.0 PL=0
MOVL C00158 V=800.0 PL=0
MOVL C00159 V=800.0 PL=0
MOVL C00160 V=800.0 PL=0
MOVL C00161 V=800.0 PL=0
MOVL C00162 V=800.0 PL=0
MOVL C00163 V=800.0 PL=0
MOVL C00164 V=800.0 PL=0
MOVL C00165 V=800.0 PL=0
MOVL C00166 V=800.0 PL=0
MOVL C00167 V=800.0 PL=0
MOVL C00168 V=800.0 PL=0
MOVL C00169 V=800.0 PL=0
MOVL C00170 V=800.0 PL=0
MOVL C00171 V=800.0 PL=0
MOVL C00172 V=800.0 PL=0
MOVL C00173 V=800.0 PL=0
MOVL C00174 V=800.0 PL=0
MOVL C00175 V=800.0 PL=0
MOVL C00176 V=800.0 PL=0
MOVL C00177 V=800.0 PL=0
MOVL C00178 V=800.0 PL=0
MOVL C00179 V=800.0 PL=0
MOVL C00180 V=800.0 PL=0
MOVL C00181 V=800.0 PL=0
MOVL C00182 V=800.0 PL=0
MOVL C00183 V=800.0 PL=0
MOVL C00184 V=800.0 PL=0
MOVL C00185 V=800.0 PL=0
MOVL C00186 V=800.0 PL=0
MOVL C00187 V=800.0 PL=0
MOVL C00188 V=800.0 PL=0
MOVL C00189 V=800.0 PL=0
MOVL C00190 V=800.0 PL=0
MOVL C00191 V=800.0 PL=0
MOVL C00192 V=800.0 PL=0
MOVL C00193 V=800.0 PL=0
MOVL C00194 V=800.0 PL=0
MOVL C00195 V=800.0 PL=0
MOVL C00196 V=800.0 PL=0
MOVL C00197 V=800.0 PL=0
MOVL C00198 V=800.0 PL=0
MOVL C00199 V=800.0 PL=0
MOVL C00200 V=800.0 PL=0
MOVL C00201 V=800.0 PL=0
MOVL C00202 V=800.0 PL=0
MOVL C00203 V=800.0 PL=0
MOVL C00204 V=800.0 PL=0
MOVL C00205 V=800.0 PL=0
MOVL C00206 V=800.0 PL=0
MOVL C00207 V=800.0 PL=0
MOVL C00208 V=800.0 PL=0
MOVL C00209 V=800.0 PL=0
MOVL C00210 V=800.0 PL=0
MOVL C00211 V=800.0 PL=0
MOVL C00212 V=800.0 PL=0
MOVL C00213 V=800.0 PL=0
MOVL C00214 V=800.0 PL=0
MOVL C00215 V=800.0 PL=0
MOVL C00216 V=800.0 PL=0
MOVL C00217 V=800.0 PL=0
MOVL C00218 V=800.0 PL=0
MOVL C00219 V=800.0 PL=0
MOVL C00220 V=800.0 PL=0
MOVL C00221 V=800.0 PL=0
MOVL C00222 V=800.0 PL=0
MOVL C00223 V=800.0 PL=0
MOVL C00224 V=800.0 PL=0
MOVL C00225 V=800.0 PL=0
MOVL C00226 V=800.0 PL=0
MOVL C00227 V=800.0 PL=0
MOVL C00228 V=800.0 PL=0
MOVL C00229 V=800.0 PL=0
MOVL C00230 V=800.0 PL=0
MOVL C00231 V=800.0 PL=0
MOVL C00232 V=800.0 PL=0
MOVL C00233 V=800.0 PL=0
MOVL C00234 V=800.0 PL=0
MOVL C00235 V=800.0 PL=0
MOVL C00236 V=800.0 PL=0
MOVL C00237 V=800.0 PL=0
MOVL C00238 V=800.0 PL=0
MOVL C00239 V=800.0 PL=0
MOVL C00240 V=800.0 PL=0
MOVL C00241 V=800.0 PL=0
MOVL C00242 V=800.0 PL=0
MOVL C00243 V=800.0 PL=0
MOVL C00244 V=800.0 PL=0
MOVL C00245 V=800.0 PL=0
MOVL C00246 V=800.0 PL=0
MOVL C00247 V=800.0 PL=0
MOVL C00248 V=800.0 PL=0
MOVL C00249 V=800.0 PL=0
MOVL C00250 V=800.0 PL=0
MOVL C00251 V=800.0 PL=0
MOVL C00252 V=800.0 PL=0
MOVL C00253 V=800.0 PL=0
MOVL C00254 V=800.0 PL=0
MOVL C00255 V=800.0 PL=0
MOVL C00256 V=800.0 PL=0
MOVL C00257 V=800.0 PL=0
MOVL C00258 V=800.0 PL=0
MOVL C00259 V=800.0 PL=0
MOVL C00260 V=800.0 PL=0
MOVL C00261 V=800.0 PL=0
MOVL C00262 V=800.0 PL=0
MOVL C00263 V=800.0 PL=0
MOVL C00264 V=800.0 PL=0
MOVL C00265 V=800.0 PL=0
MOVL C00266 V=800.0 PL=0
MOVL C00267 V=800.0 PL=0
MOVL C00268 V=800.0 PL=0
MOVL C00269 V=800.0 PL=0
MOVL C00270 V=800.0 PL=0
MOVL C00271 V=800.0 PL=0
MOVL C00272 V=800.0 PL=0
MOVL C00273 V=800.0 PL=0
MOVL C00274 V=800.0 PL=0
MOVL C00275 V=800.0 PL=0
MOVL C00276 V=800.0 PL=0
MOVL C00277 V=800.0 PL=0
MOVL C00278 V=800.0 PL=0
MOVL C00279 V=800.0 PL=0
MOVL C00280 V=800.0 PL=0
MOVL C00281 V=800.0 PL=0
MOVL C00282 V=800.0 PL=0
MOVL C00283 V=800.0 PL=0
MOVL C00284 V=800.0 PL=0
MOVL C00285 V=800.0 PL=0
MOVL C00286 V=800.0 PL=0
MOVL C00287 V=800.0 PL=0
MOVL C00288 V=800.0 PL=0
MOVL C00289 V=800.0 PL=0
MOVL C00290 V=800.0 PL=0
MOVL C00291 V=800.0 PL=0
MOVL C00292 V=800.0 PL=0
MOVL C00293 V=800.0 PL=0
MOVL C00294 V=800.0 PL=0
MOVL C00295 V=800.0 PL=0
MOVL C00296 V=800.0 PL=0
MOVL C00297 V=800.0 PL=0
MOVL C00298 V=800.0 PL=0
MOVL C00299 V=800.0 PL=0
MOVL C00300 V=800.0 PL=0
MOVL C00301 V=800.0 PL=0
MOVL C00302 V=800.0 PL=0
MOVL C00303 V=800.0 PL=0
MOVL C00304 V=800.0 PL=0
MOVL C00305 V=800.0 PL=0
MOVL C00306 V=800.0 PL=0
MOVL C00307 V=800.0 PL=0
MOVL C00308 V=800.0 PL=0
MOVL C00309 V=800.0 PL=0
MOVL C00310 V=800.0 PL=0
MOVL C00311 V=800.0 PL=0
MOVL C00312 V=800.0 PL=0
MOVL C00313 V=800.0 PL=0
MOVL C00314 V=800.0 PL=0
MOVL C00315 V=800.0 PL=0
MOVL C00316 V=800.0 PL=0
MOVL C00317 V=800.0 PL=0
MOVL C00318 V=800.0 PL=0
MOVL C00319 V=800.0 PL=0
MOVL C00320 V=800.0 PL=0
MOVL C00321 V=800.0 PL=0
MOVL C00322 V=800.0 PL=0
MOVL C00323 V=800.0 PL=0
MOVL C00324 V=800.0 PL=0
MOVL C00325 V=800.0 PL=0
MOVL C00326 V=800.0 PL=0
MOVL C00327 V=800.0 PL=0
MOVL C00328 V=800.0 PL=0
MOVL C00329 V=800.0 PL=0
MOVL C00330 V=800.0 PL=0
MOVL C00331 V=800.0 PL=0
MOVL C00332 V=800.0 PL=0
MOVL C00333 V=800.0 PL=0
MOVL C00334 V=800.0 PL=0
MOVL C00335 V=800.0 PL=0
MOVL C00336 V=800.0 PL=0
MOVL C00337 V=800.0 PL=0
MOVL C00338 V=800.0 PL=0
MOVL C00339 V=800.0 PL=0
MOVL C00340 V=800.0 PL=0
MOVL C00341 V=800.0 PL=0
MOVL C00342 V=800.0 PL=0
MOVL C00343 V=800.0 PL=0
MOVL C00344 V=800.0 PL=0
MOVL C00345 V=800.0 PL=0
MOVL C00346 V=800.0 PL=0
MOVL C00347 V=800.0 PL=0
MOVL C00348 V=800.0 PL=0
MOVL C00349 V=800.0 PL=0
MOVL C00350 V=800.0 PL=0
MOVL C00351 V=800.0 PL=0
MOVL C00352 V=800.0 PL=0
MOVL C00353 V=800.0 PL=0
MOVL C00354 V=800.0 PL=0
MOVL C00355 V=800.0 PL=0
MOVL C00356 V=800.0 PL=0
MOVL C00357 V=800.0 PL=0
MOVL C00358 V=800.0 PL=0
MOVL C00359 V=800.0 PL=0
MOVL C00360 V=800.0 PL=0
MOVL C00361 V=800.0 PL=0
MOVL C00362 V=800.0 PL=0
MOVL C00363 V=800.0 PL=0
MOVL C00364 V=800.0 PL=0
MOVL C00365 V=800.0 PL=0
MOVL C00366 V=800.0 PL=0
MOVL C00367 V=800.0 PL=0
MOVL C00368 V=800.0 PL=0
MOVL C00369 V=800.0 PL=0
MOVL C00370 V=800.0 PL=0
MOVL C00371 V=800.0 PL=0
MOVL C00372 V=800.0 PL=0
MOVL C00373 V=800.0 PL=0
MOVL C00374 V=800.0 PL=0
MOVL C00375 V=800.0 PL=0
MOVL C00376 V=800.0 PL=0
MOVL C00377 V=800.0 PL=0
MOVL C00378 V=800.0 PL=0
MOVL C00379 V=800.0 PL=0
MOVL C00380 V=800.0 PL=0
MOVL C00381 V=800.0 PL=0
MOVL C00382 V=800.0 PL=0
MOVL C00383 V=800.0 PL=0
MOVL C00384 V=800.0 PL=0
MOVL C00385 V=800.0 PL=0
MOVL C00386 V=800.0 PL=0
MOVL C00387 V=800.0 PL=0
MOVL C00388 V=800.0 PL=0
MOVL C00389 V=800.0 PL=0
MOVL C00390 V=800.0 PL=0
MOVL C00391 V=800.0 PL=0
MOVL C00392 V=800.0 PL=0
MOVL C00393 V=800.0 PL=0
MOVL C00394 V=800.0 PL=0
MOVL C00395 V=800.0 PL=0
MOVL C00396 V=800.0 PL=0
MOVL C00397 V=800.0 PL=0
MOVL C00398 V=800.0 PL=0
MOVL C00399 V=800.0 PL=0
MOVL C00400 V=800.0 PL=0
MOVL C00401 V=800.0 PL=0
MOVL C00402 V=800.0 PL=0
MOVL C00403 V=800.0 PL=0
MOVL C00404 V=800.0 PL=0
MOVL C00405 V=800.0 PL=0
MOVL C00406 V=800.0 PL=0
MOVL C00407 V=800.0 PL=0
MOVL C00408 V=800.0 PL=0
MOVL C00409 V=800.0 PL=0
MOVL C00410 V=800.0 PL=0
MOVL C00411 V=800.0 PL=0
MOVL C00412 V=800.0 PL=0
MOVL C00413 V=800.0 PL=0
MOVL C00414 V=800.0 PL=0
MOVL C00415 V=800.0 PL=0
MOVL C00416 V=800.0 PL=0
MOVL C00417 V=800.0 PL=0
MOVL C00418 V=800.0 PL=0
MOVL C00419 V=800.0 PL=0
MOVL C00420 V=800.0 PL=0
MOVL C00421 V=800.0 PL=0
MOVL C00422 V=800.0 PL=0
MOVL C00423 V=800.0 PL=0
MOVL C00424 V=800.0 PL=0
MOVL C00425 V=800.0 PL=0
MOVL C00426 V=800.0 PL=0
MOVL C00427 V=800.0 PL=0
MOVL C00428 V=800.0 PL=0
MOVL C00429 V=800.0 PL=0
MOVL C00430 V=800.0 PL=0
MOVL C00431 V=800.0 PL=0
MOVL C00432 V=800.0 PL=0
MOVL C00433 V=800.0 PL=0
MOVL C00434 V=800.0 PL=0
MOVL C00435 V=800.0 PL=0
MOVL C00436 V=800.0 PL=0
MOVL C00437 V=800.0 PL=0
MOVL C00438 V=800.0 PL=0
MOVL C00439 V=800.0 PL=0
MOVL C00440 V=800.0 PL=0
MOVL C00441 V=800.0 PL=0
MOVL C00442 V=800.0 PL=0
MOVL C00443 V=800.0 PL=0
MOVL C00444 V=800.0 PL=0
MOVL C00445 V=800.0 PL=0
MOVL C00446 V=800.0 PL=0
MOVL C00447 V=800.0 PL=0
MOVL C00448 V=800.0 PL=0
MOVL C00449 V=800.0 PL=0
MOVL C00450 V=800.0 PL=0
MOVL C00451 V=800.0 PL=0
MOVL C00452 V=800.0 PL=0
MOVL C00453 V=800.0 PL=0
MOVL C00454 V=800.0 PL=0
MOVL C00455 V=800.0 PL=0
MOVL C00456 V=800.0 PL=0
MOVL C00457 V=800.0 PL=0
MOVL C00458 V=800.0 PL=0
MOVL C00459 V=800.0 PL=0
MOVL C00460 V=800.0 PL=0
MOVL C00461 V=800.0 PL=0
MOVL C00462 V=800.0 PL=0
MOVL C00463 V=800.0 PL=0
MOVL C00464 V=800.0 PL=0
MOVL C00465 V=800.0 PL=0
MOVL C00466 V=800.0 PL=0
MOVL C00467 V=800.0 PL=0
MOVL C00468 V=800.0 PL=0
MOVL C00469 V=800.0 PL=0
MOVL C00470 V=800.0 PL=0
MOVL C00471 V=800.0 PL=0
MOVL C00472 V=800.0 PL=0
MOVL C00473 V=800.0 PL=0
MOVL C00474 V=800.0 PL=0
MOVL C00475 V=800.0 PL=0
MOVL C00476 V=800.0 PL=0
MOVL C00477 V=800.0 PL=0
MOVL C00478 V=800.0 PL=0
MOVL C00479 V=800.0 PL=0
MOVL C00480 V=800.0 PL=0
MOVL C00481 V=800.0 PL=0
MOVL C00482 V=800.0 PL=0
MOVL C00483 V=800.0 PL=0
MOVL C00484 V=800.0 PL=0
MOVL C00485 V=800.0 PL=0
MOVL C00486 V=800.0 PL=0
MOVL C00487 V=800.0 PL=0
MOVL C00488 V=800.0 PL=0
MOVL C00489 V=800.0 PL=0
MOVL C00490 V=800.0 PL=0
MOVL C00491 V=800.0 PL=0
MOVL C00492 V=800.0 PL=0
MOVL C00493 V=800.0 PL=0
MOVL C00494 V=800.0 PL=0
MOVL C00495 V=800.0 PL=0
MOVL C00496 V=800.0 PL=0
MOVL C00497 V=800.0 PL=0
MOVL C00498 V=800.0 PL=0
MOVL C00499 V=800.0 PL=0
MOVL C00500 V=800.0 PL=0
MOVL C00501 V=800.0 PL=0
MOVL C00502 V=800.0 PL=0
MOVL C00503 V=800.0 PL=0
MOVL C00504 V=800.0 PL=0
MOVL C00505 V=800.0 PL=0
MOVL C00506 V=800.0 PL=0
MOVL C00507 V=800.0 PL=0
MOVL C00508 V=800.0 PL=0
MOVL C00509 V=800.0 PL=0
MOVL C00510 V=800.0 PL=0
MOVL C00511 V=800.0 PL=0
MOVL C00512 V=800.0 PL=0
MOVL C00513 V=800.0 PL=0
MOVL C00514 V=800.0 PL=0
MOVL C00515 V=800.0 PL=0
MOVL C00516 V=800.0 PL=0
MOVL C00517 V=800.0 PL=0
MOVL C00518 V=800.0 PL=0
MOVL C00519 V=800.0 PL=0
MOVL C00520 V=800.0 PL=0
MOVL C00521 V=800.0 PL=0
MOVL C00522 V=800.0 PL=0
MOVL C00523 V=800.0 PL=0
MOVL C00524 V=800.0 PL=0
MOVL C00525 V=800.0 PL=0
MOVL C00526 V=800.0 PL=0
MOVL C00527 V=800.0 PL=0
MOVL C00528 V=800.0 PL=0
MOVL C00529 V=800.0 PL=0
MOVL C00530 V=800.0 PL=0
MOVL C00531 V=800.0 PL=0
MOVL C00532 V=800.0 PL=0
MOVL C00533 V=800.0 PL=0
MOVL C00534 V=800.0 PL=0
MOVL C00535 V=800.0 PL=0
MOVL C00536 V=800.0 PL=0
MOVL C00537 V=800.0 PL=0
MOVL C00538 V=800.0 PL=0
MOVL C00539 V=800.0 PL=0
MOVL C00540 V=800.0 PL=0
MOVL C00541 V=800.0 PL=0
MOVL C00542 V=800.0 PL=0
MOVL C00543 V=800.0 PL=0
MOVL C00544 V=800.0 PL=0
MOVL C00545 V=800.0 PL=0
MOVL C00546 V=800.0 PL=0
MOVL C00547 V=800.0 PL=0
MOVL C00548 V=800.0 PL=0
MOVL C00549 V=800.0 PL=0
MOVL C00550 V=800.0 PL=0
MOVL C00551 V=800.0 PL=0
MOVL C00552 V=800.0 PL=0
MOVL C00553 V=800.0 PL=0
MOVL C00554 V=800.0 PL=0
MOVL C00555 V=800.0 PL=0
MOVL C00556 V=800.0 PL=0
MOVL C00557 V=800.0 PL=0
MOVL C00558 V=800.0 PL=0
MOVL C00559 V=800.0 PL=0
MOVL C00560 V=800.0 PL=0
MOVL C00561 V=800.0 PL=0
MOVL C00562 V=800.0 PL=0
MOVL C00563 V=800.0 PL=0
MOVL C00564 V=800.0 PL=0
MOVL C00565 V=800.0 PL=0
MOVL C00566 V=800.0 PL=0
MOVL C00567 V=800.0 PL=0
MOVL C00568 V=800.0 PL=0
MOVL C00569 V=800.0 PL=0
MOVL C00570 V=800.0 PL=0
MOVL C00571 V=800.0 PL=0
MOVL C00572 V=800.0 PL=0
MOVL C00573 V=800.0 PL=0
MOVL C00574 V=800.0 PL=0
MOVL C00575 V=800.0 PL=0
MOVL C00576 V=800.0 PL=0
MOVL C00577 V=800.0 PL=0
MOVL C00578 V=800.0 PL=0
MOVL C00579 V=800.0 PL=0
MOVL C00580 V=800.0 PL=0
MOVL C00581 V=800.0 PL=0
MOVL C00582 V=800.0 PL=0
MOVL C00583 V=800.0 PL=0
MOVL C00584 V=800.0 PL=0
MOVL C00585 V=800.0 PL=0
MOVL C00586 V=800.0 PL=0
MOVL C00587 V=800.0 PL=0
MOVL C00588 V=800.0 PL=0
MOVL C00589 V=800.0 PL=0
MOVL C00590 V=800.0 PL=0
MOVL C00591 V=800.0 PL=0
MOVL C00592 V=800.0 PL=0
MOVL C00593 V=800.0 PL=0
MOVL C00594 V=800.0 PL=0
MOVL C00595 V=800.0 PL=0
MOVL C00596 V=800.0 PL=0
MOVL C00597 V=800.0 PL=0
MOVL C00598 V=800.0 PL=0
MOVL C00599 V=800.0 PL=0
MOVL C00600 V=800.0 PL=0
MOVL C00601 V=800.0 PL=0
MOVL C00602 V=800.0 PL=0
MOVL C00603 V=800.0 PL=0
MOVL C00604 V=800.0 PL=0
MOVL C00605 V=800.0 PL=0
MOVL C00606 V=800.0 PL=0
MOVL C00607 V=800.0 PL=0
MOVL C00608 V=800.0 PL=0
MOVL C00609 V=800.0 PL=0
MOVL C00610 V=800.0 PL=0
MOVL C00611 V=800.0 PL=0
MOVL C00612 V=800.0 PL=0
MOVL C00613 V=800.0 PL=0
MOVL C00614 V=800.0 PL=0
MOVL C00615 V=800.0 PL=0
MOVL C00616 V=800.0 PL=0
MOVL C00617 V=800.0 PL=0
MOVL C00618 V=800.0 PL=0
MOVL C00619 V=800.0 PL=0
MOVL C00620 V=800.0 PL=0
MOVL C00621 V=800.0 PL=0
MOVL C00622 V=800.0 PL=0
MOVL C00623 V=800.0 PL=0
MOVL C00624 V=800.0 PL=0
MOVL C00625 V=800.0 PL=0
MOVL C00626 V=800.0 PL=0
MOVL C00627 V=800.0 PL=0
MOVL C00628 V=800.0 PL=0
MOVL C00629 V=800.0 PL=0
MOVL C00630 V=800.0 PL=0
MOVL C00631 V=800.0 PL=0
MOVL C00632 V=800.0 PL=0
MOVL C00633 V=800.0 PL=0
MOVL C00634 V=800.0 PL=0
MOVL C00635 V=800.0 PL=0
MOVL C00636 V=800.0 PL=0
MOVL C00637 V=800.0 PL=0
MOVL C00638 V=800.0 PL=0
MOVL C00639 V=800.0 PL=0
MOVL C00640 V=800.0 PL=0
MOVL C00641 V=800.0 PL=0
MOVL C00642 V=800.0 PL=0
MOVL C00643 V=800.0 PL=0
MOVL C00644 V=800.0 PL=0
MOVL C00645 V=800.0 PL=0
MOVL C00646 V=800.0 PL=0
MOVL C00647 V=800.0 PL=0
MOVL C00648 V=800.0 PL=0
MOVL C00649 V=800.0 PL=0
MOVL C00650 V=800.0 PL=0
MOVL C00651 V=800.0 PL=0
MOVL C00652 V=800.0 PL=0
MOVL C00653 V=800.0 PL=0
MOVL C00654 V=800.0 PL=0
MOVL C00655 V=800.0 PL=0
MOVL C00656 V=800.0 PL=0
MOVL C00657 V=800.0 PL=0
MOVL C00658 V=800.0 PL=0
MOVL C00659 V=800.0 PL=0
MOVL C00660 V=800.0 PL=0
MOVL C00661 V=800.0 PL=0
MOVL C00662 V=800.0 PL=0
MOVL C00663 V=800.0 PL=0
MOVL C00664 V=800.0 PL=0
MOVL C00665 V=800.0 PL=0
MOVL C00666 V=800.0 PL=0
MOVL C00667 V=800.0 PL=0
MOVL C00668 V=800.0 PL=0
MOVL C00669 V=800.0 PL=0
MOVL C00670 V=800.0 PL=0
MOVL C00671 V=800.0 PL=0
MOVL C00672 V=800.0 PL=0
MOVL C00673 V=800.0 PL=0
MOVL C00674 V=800.0 PL=0
MOVL C00675 V=800.0 PL=0
MOVL C00676 V=800.0 PL=0
MOVL C00677 V=800.0 PL=0
MOVL C00678 V=800.0 PL=0
MOVL C00679 V=800.0 PL=0
MOVL C00680 V=800.0 PL=0
MOVL C00681 V=800.0 PL=0
MOVL C00682 V=800.0 PL=0
MOVL C00683 V=800.0 PL=0
MOVL C00684 V=800.0 PL=0
MOVL C00685 V=800.0 PL=0
MOVL C00686 V=800.0 PL=0
MOVL C00687 V=800.0 PL=0
MOVL C00688 V=800.0 PL=0
MOVL C00689 V=800.0 PL=0
MOVL C00690 V=800.0 PL=0
MOVL C00691 V=800.0 PL=0
MOVL C00692 V=800.0 PL=0
MOVL C00693 V=800.0 PL=0
MOVL C00694 V=800.0 PL=0
MOVL C00695 V=800.0 PL=0
MOVL C00696 V=800.0 PL=0
MOVL C00697 V=800.0 PL=0
MOVL C00698 V=800.0 PL=0
MOVL C00699 V=800.0 PL=0
MOVL C00700 V=800.0 PL=0
MOVL C00701 V=800.0 PL=0
MOVL C00702 V=800.0 PL=0
MOVL C00703 V=800.0 PL=0
MOVL C00704 V=800.0 PL=0
MOVL C00705 V=800.0 PL=0
MOVL C00706 V=800.0 PL=0
MOVL C00707 V=800.0 PL=0
MOVL C00708 V=800.0 PL=0
MOVL C00709 V=800.0 PL=0
MOVL C00710 V=800.0 PL=0
MOVL C00711 V=800.0 PL=0
MOVL C00712 V=800.0 PL=0
MOVL C00713 V=800.0 PL=0
MOVL C00714 V=800.0 PL=0
MOVL C00715 V=800.0 PL=0
MOVL C00716 V=800.0 PL=0
MOVL C00717 V=800.0 PL=0
MOVL C00718 V=800.0 PL=0
MOVL C00719 V=800.0 PL=0
MOVL C00720 V=800.0 PL=0
MOVL C00721 V=800.0 PL=0
MOVL C00722 V=800.0 PL=0
MOVL C00723 V=800.0 PL=0
MOVL C00724 V=800.0 PL=0
MOVL C00725 V=800.0 PL=0
MOVL C00726 V=800.0 PL=0
MOVL C00727 V=800.0 PL=0
MOVL C00728 V=800.0 PL=0
MOVL C00729 V=800.0 PL=0
MOVL C00730 V=800.0 PL=0
MOVL C00731 V=800.0 PL=0
MOVL C00732 V=800.0 PL=0
MOVL C00733 V=800.0 PL=0
MOVL C00734 V=800.0 PL=0
MOVL C00735 V=800.0 PL=0
MOVL C00736 V=800.0 PL=0
MOVL C00737 V=800.0 PL=0
MOVL C00738 V=800.0 PL=0
MOVL C00739 V=800.0 PL=0
MOVL C00740 V=800.0 PL=0
MOVL C00741 V=800.0 PL=0
MOVL C00742 V=800.0 PL=0
MOVL C00743 V=800.0 PL=0
MOVL C00744 V=800.0 PL=0
MOVL C00745 V=800.0 PL=0
MOVL C00746 V=800.0 PL=0
MOVL C00747 V=800.0 PL=0
MOVL C00748 V=800.0 PL=0
MOVL C00749 V=800.0 PL=0
MOVL C00750 V=800.0 PL=0
MOVL C00751 V=800.0 PL=0
MOVL C00752 V=800.0 PL=0
MOVL C00753 V=800.0 PL=0
MOVL C00754 V=800.0 PL=0
MOVL C00755 V=800.0 PL=0
MOVL C00756 V=800.0 PL=0
MOVL C00757 V=800.0 PL=0
MOVL C00758 V=800.0 PL=0
MOVL C00759 V=800.0 PL=0
MOVL C00760 V=800.0 PL=0
MOVL C00761 V=800.0 PL=0
MOVL C00762 V=800.0 PL=0
MOVL C00763 V=800.0 PL=0
MOVL C00764 V=800.0 PL=0
MOVL C00765 V=800.0 PL=0
MOVL C00766 V=800.0 PL=0
MOVL C00767 V=800.0 PL=0
MOVL C00768 V=800.0 PL=0
MOVL C00769 V=800.0 PL=0
MOVL C00770 V=800.0 PL=0
MOVL C00771 V=800.0 PL=0
MOVL C00772 V=800.0 PL=0
MOVL C00773 V=800.0 PL=0
MOVL C00774 V=800.0 PL=0
MOVL C00775 V=800.0 PL=0
MOVL C00776 V=800.0 PL=0
MOVL C00777 V=800.0 PL=0
MOVL C00778 V=800.0 PL=0
MOVL C00779 V=800.0 PL=0
MOVL C00780 V=800.0 PL=0
MOVL C00781 V=800.0 PL=0
MOVL C00782 V=800.0 PL=0
MOVL C00783 V=800.0 PL=0
MOVL C00784 V=800.0 PL=0
MOVL C00785 V=800.0 PL=0
MOVL C00786 V=800.0 PL=0
MOVL C00787 V=800.0 PL=0
MOVL C00788 V=800.0 PL=0
MOVL C00789 V=800.0 PL=0
MOVL C00790 V=800.0 PL=0
MOVL C00791 V=800.0 PL=0
MOVL C00792 V=800.0 PL=0
MOVL C00793 V=800.0 PL=0
MOVL C00794 V=800.0 PL=0
MOVL C00795 V=800.0 PL=0
MOVL C00796 V=800.0 PL=0
MOVL C00797 V=800.0 PL=0
MOVL C00798 V=800.0 PL=0
MOVL C00799 V=800.0 PL=0
MOVL C00800 V=800.0 PL=0
MOVL C00801 V=800.0 PL=0
MOVL C00802 V=800.0 PL=0
MOVL C00803 V=800.0 PL=0
MOVL C00804 V=800.0 PL=0
MOVL C00805 V=800.0 PL=0
MOVL C00806 V=800.0 PL=0
MOVL C00807 V=800.0 PL=0
MOVL C00808 V=800.0 PL=0
MOVL C00809 V=800.0 PL=0
MOVL C00810 V=800.0 PL=0
MOVL C00811 V=800.0 PL=0
MOVL C00812 V=800.0 PL=0
MOVL C00813 V=800.0 PL=0
MOVL C00814 V=800.0 PL=0
MOVL C00815 V=800.0 PL=0
MOVL C00816 V=800.0 PL=0
MOVL C00817 V=800.0 PL=0
MOVL C00818 V=800.0 PL=0
MOVL C00819 V=800.0 PL=0
MOVL C00820 V=800.0 PL=0
MOVL C00821 V=800.0 PL=0
MOVL C00822 V=800.0 PL=0
MOVL C00823 V=800.0 PL=0
MOVL C00824 V=800.0 PL=0
MOVL C00825 V=800.0 PL=0
MOVL C00826 V=800.0 PL=0
MOVL C00827 V=800.0 PL=0
MOVL C00828 V=800.0 PL=0
MOVL C00829 V=800.0 PL=0
MOVL C00830 V=800.0 PL=0
MOVL C00831 V=800.0 PL=0
MOVL C00832 V=800.0 PL=0
MOVL C00833 V=800.0 PL=0
MOVL C00834 V=800.0 PL=0
MOVL C00835 V=800.0 PL=0
MOVL C00836 V=800.0 PL=0
MOVL C00837 V=800.0 PL=0
MOVL C00838 V=800.0 PL=0
MOVL C00839 V=800.0 PL=0
MOVL C00840 V=800.0 PL=0
MOVL C00841 V=800.0 PL=0
MOVL C00842 V=800.0 PL=0
MOVL C00843 V=800.0 PL=0
MOVL C00844 V=800.0 PL=0
MOVL C00845 V=800.0 PL=0
MOVL C00846 V=800.0 PL=0
MOVL C00847 V=800.0 PL=0
MOVL C00848 V=800.0 PL=0
MOVL C00849 V=800.0 PL=0
MOVL C00850 V=800.0 PL=0
MOVL C00851 V=800.0 PL=0
MOVL C00852 V=800.0 PL=0
MOVL C00853 V=800.0 PL=0
MOVL C00854 V=800.0 PL=0
MOVL C00855 V=800.0 PL=0
MOVL C00856 V=800.0 PL=0
MOVL C00857 V=800.0 PL=0
MOVL C00858 V=800.0 PL=0
MOVL C00859 V=800.0 PL=0
MOVL C00860 V=800.0 PL=0
MOVL C00861 V=800.0 PL=0
MOVL C00862 V=800.0 PL=0
MOVL C00863 V=800.0 PL=0
MOVL C00864 V=800.0 PL=0
MOVL C00865 V=800.0 PL=0
MOVL C00866 V=800.0 PL=0
MOVL C00867 V=800.0 PL=0
MOVL C00868 V=800.0 PL=0
MOVL C00869 V=800.0 PL=0
MOVL C00870 V=800.0 PL=0
MOVL C00871 V=800.0 PL=0
MOVL C00872 V=800.0 PL=0
MOVL C00873 V=800.0 PL=0
MOVL C00874 V=800.0 PL=0
MOVL C00875 V=800.0 PL=0
MOVL C00876 V=800.0 PL=0
MOVL C00877 V=800.0 PL=0
MOVL C00878 V=800.0 PL=0
MOVL C00879 V=800.0 PL=0
MOVL C00880 V=800.0 PL=0
MOVL C00881 V=800.0 PL=0
MOVL C00882 V=800.0 PL=0
MOVL C00883 V=800.0 PL=0
MOVL C00884 V=800.0 PL=0
MOVL C00885 V=800.0 PL=0
MOVL C00886 V=800.0 PL=0
MOVL C00887 V=800.0 PL=0
MOVL C00888 V=800.0 PL=0
MOVL C00889 V=800.0 PL=0
MOVL C00890 V=800.0 PL=0
MOVL C00891 V=800.0 PL=0
MOVL C00892 V=800.0 PL=0
MOVL C00893 V=800.0 PL=0
MOVL C00894 V=800.0 PL=0
MOVL C00895 V=800.0 PL=0
MOVL C00896 V=800.0 PL=0
MOVL C00897 V=800.0 PL=0
MOVL C00898 V=800.0 PL=0
MOVL C00899 V=800.0 PL=0
MOVL C00900 V=800.0 PL=0
MOVL C00901 V=800.0 PL=0
MOVL C00902 V=800.0 PL=0
MOVL C00903 V=800.0 PL=0
MOVL C00904 V=800.0 PL=0
MOVL C00905 V=800.0 PL=0
MOVL C00906 V=800.0 PL=0
MOVL C00907 V=800.0 PL=0
MOVL C00908 V=800.0 PL=0
MOVL C00909 V=800.0 PL=0
MOVL C00910 V=800.0 PL=0
MOVL C00911 V=800.0 PL=0
MOVL C00912 V=800.0 PL=0
MOVL C00913 V=800.0 PL=0
MOVL C00914 V=800.0 PL=0
MOVL C00915 V=800.0 PL=0
MOVL C00916 V=800.0 PL=0
MOVL C00917 V=800.0 PL=0
MOVL C00918 V=800.0 PL=0
MOVL C00919 V=800.0 PL=0
MOVL C00920 V=800.0 PL=0
MOVL C00921 V=800.0 PL=0
MOVL C00922 V=800.0 PL=0
MOVL C00923 V=800.0 PL=0
MOVL C00924 V=800.0 PL=0
MOVL C00925 V=800.0 PL=0
MOVL C00926 V=800.0 PL=0
MOVL C00927 V=800.0 PL=0
MOVL C00928 V=800.0 PL=0
MOVL C00929 V=800.0 PL=0
MOVL C00930 V=800.0 PL=0
MOVL C00931 V=800.0 PL=0
MOVL C00932 V=800.0 PL=0
MOVL C00933 V=800.0 PL=0
MOVL C00934 V=800.0 PL=0
MOVL C00935 V=800.0 PL=0
MOVL C00936 V=800.0 PL=0
MOVL C00937 V=800.0 PL=0
MOVL C00938 V=800.0 PL=0
MOVL C00939 V=800.0 PL=0
MOVL C00940 V=800.0 PL=0
MOVL C00941 V=800.0 PL=0
MOVL C00942 V=800.0 PL=0
MOVL C00943 V=800.0 PL=0
MOVL C00944 V=800.0 PL=0
MOVL C00945 V=800.0 PL=0
MOVL C00946 V=800.0 PL=0
MOVL C00947 V=800.0 PL=0
MOVL C00948 V=800.0 PL=0
MOVL C00949 V=800.0 PL=0
MOVL C00950 V=800.0 PL=0
MOVL C00951 V=800.0 PL=0
MOVL C00952 V=800.0 PL=0
MOVL C00953 V=800.0 PL=0
MOVL C00954 V=800.0 PL=0
MOVL C00955 V=800.0 PL=0
MOVL C00956 V=800.0 PL=0
MOVL C00957 V=800.0 PL=0
MOVL C00958 V=800.0 PL=0
MOVL C00959 V=800.0 PL=0
MOVL C00960 V=800.0 PL=0
MOVL C00961 V=800.0 PL=0
MOVL C00962 V=800.0 PL=0
MOVL C00963 V=800.0 PL=0
MOVL C00964 V=800.0 PL=0
MOVL C00965 V=800.0 PL=0
MOVL C00966 V=800.0 PL=0
MOVL C00967 V=800.0 PL=0
MOVL C00968 V=800.0 PL=0
MOVL C00969 V=800.0 PL=0
MOVL C00970 V=800.0 PL=0
MOVL C00971 V=800.0 PL=0
MOVL C00972 V=800.0 PL=0
MOVL C00973 V=800.0 PL=0
MOVL C00974 V=800.0 PL=0
MOVL C00975 V=800.0 PL=0
MOVL C00976 V=800.0 PL=0
MOVL C00977 V=800.0 PL=0
MOVL C00978 V=800.0 PL=0
MOVL C00979 V=800.0 PL=0
MOVL C00980 V=800.0 PL=0
MOVL C00981 V=800.0 PL=0
MOVL C00982 V=800.0 PL=0
MOVL C00983 V=800.0 PL=0
MOVL C00984 V=800.0 PL=0
MOVL C00985 V=800.0 PL=0
MOVL C00986 V=800.0 PL=0
MOVL C00987 V=800.0 PL=0
MOVL C00988 V=800.0 PL=0
MOVL C00989 V=800.0 PL=0
MOVL C00990 V=800.0 PL=0
MOVL C00991 V=800.0 PL=0
MOVL C00992 V=800.0 PL=0
MOVL C00993 V=800.0 PL=0
MOVL C00994 V=800.0 PL=0
MOVL C00995 V=800.0 PL=0
MOVL C00996 V=800.0 PL=0
MOVL C00997 V=800.0 PL=0
MOVL C00998 V=800.0 PL=0
MOVL C00999 V=800.0 PL=0
MOVL C01000 V=800.0 PL=0
MOVL C01001 V=800.0 PL=0
MOVL C01002 V=800.0 PL=0
MOVL C01003 V=800.0 PL=0
MOVL C01004 V=800.0 PL=0
MOVL C01005 V=800.0 PL=0
MOVL C01006 V=800.0 PL=0
MOVL C01007 V=800.0 PL=0
MOVL C01008 V=800.0 PL=0
MOVL C01009 V=800.0 PL=0
MOVL C01010 V=800.0 PL=0
MOVL C01011 V=800.0 PL=0
MOVL C01012 V=800.0 PL=0
MOVL C01013 V=800.0 PL=0
MOVL C01014 V=800.0 PL=0
MOVL C01015 V=800.0 PL=0
MOVL C01016 V=800.0 PL=0
MOVL C01017 V=800.0 PL=0
MOVL C01018 V=800.0 PL=0
MOVL C01019 V=800.0 PL=0
MOVL C01020 V=800.0 PL=0
MOVL C01021 V=800.0 PL=0
MOVL C01022 V=800.0 PL=0
MOVL C01023 V=800.0 PL=0
MOVL C01024 V=800.0 PL=0
MOVL C01025 V=800.0 PL=0
MOVL C01026 V=800.0 PL=0
MOVL C01027 V=800.0 PL=0
MOVL C01028 V=800.0 PL=0
MOVL C01029 V=800.0 PL=0
MOVL C01030 V=800.0 PL=0
MOVL C01031 V=800.0 PL=0
MOVL C01032 V=800.0 PL=0
MOVL C01033 V=800.0 PL=0
MOVL C01034 V=800.0 PL=0
MOVL C01035 V=800.0 PL=0
MOVL C01036 V=800.0 PL=0
MOVL C01037 V=800.0 PL=0
MOVL C01038 V=800.0 PL=0
MOVL C01039 V=800.0 PL=0
MOVL C01040 V=800.0 PL=0
MOVL C01041 V=800.0 PL=0
MOVL C01042 V=800.0 PL=0
MOVL C01043 V=800.0 PL=0
MOVL C01044 V=800.0 PL=0
MOVL C01045 V=800.0 PL=0
MOVL C01046 V=800.0 PL=0
MOVL C01047 V=800.0 PL=0
MOVL C01048 V=800.0 PL=0
MOVL C01049 V=800.0 PL=0
MOVL C01050 V=800.0 PL=0
MOVL C01051 V=800.0 PL=0
MOVL C01052 V=800.0 PL=0
MOVL C01053 V=800.0 PL=0
MOVL C01054 V=800.0 PL=0
MOVL C01055 V=800.0 PL=0
MOVL C01056 V=800.0 PL=0
MOVL C01057 V=800.0 PL=0
MOVL C01058 V=800.0 PL=0
MOVL C01059 V=800.0 PL=0
MOVL C01060 V=800.0 PL=0
MOVL C01061 V=800.0 PL=0
MOVL C01062 V=800.0 PL=0
MOVL C01063 V=800.0 PL=0
MOVL C01064 V=800.0 PL=0
MOVL C01065 V=800.0 PL=0
MOVL C01066 V=800.0 PL=0
MOVL C01067 V=800.0 PL=0
MOVL C01068 V=800.0 PL=0
MOVL C01069 V=800.0 PL=0
MOVL C01070 V=800.0 PL=0
MOVL C01071 V=800.0 PL=0
MOVL C01072 V=800.0 PL=0
MOVL C01073 V=800.0 PL=0
MOVL C01074 V=800.0 PL=0
MOVL C01075 V=800.0 PL=0
MOVL C01076 V=800.0 PL=0
MOVL C01077 V=800.0 PL=0
MOVL C01078 V=800.0 PL=0
MOVL C01079 V=800.0 PL=0
MOVL C01080 V=800.0 PL=0
MOVL C01081 V=800.0 PL=0
MOVL C01082 V=800.0 PL=0
MOVL C01083 V=800.0 PL=0
MOVL C01084 V=800.0 PL=0
MOVL C01085 V=800.0 PL=0
MOVL C01086 V=800.0 PL=0
MOVL C01087 V=800.0 PL=0
MOVL C01088 V=800.0 PL=0
MOVL C01089 V=800.0 PL=0
MOVL C01090 V=800.0 PL=0
MOVL C01091 V=800.0 PL=0
MOVL C01092 V=800.0 PL=0
MOVL C01093 V=800.0 PL=0
MOVL C01094 V=800.0 PL=0
MOVL C01095 V=800.0 PL=0
MOVL C01096 V=800.0 PL=0
MOVL C01097 V=800.0 PL=0
MOVL C01098 V=800.0 PL=0
MOVL C01099 V=800.0 PL=0
MOVL C01100 V=800.0 PL=0
MOVL C01101 V=800.0 PL=0
MOVL C01102 V=800.0 PL=0
MOVL C01103 V=800.0 PL=0
MOVL C01104 V=800.0 PL=0
MOVL C01105 V=800.0 PL=0
MOVL C01106 V=800.0 PL=0
MOVL C01107 V=800.0 PL=0
MOVL C01108 V=800.0 PL=0
MOVL C01109 V=800.0 PL=0
MOVL C01110 V=800.0 PL=0
MOVL C01111 V=800.0 PL=0
MOVL C01112 V=800.0 PL=0
MOVL C01113 V=800.0 PL=0
MOVL C01114 V=800.0 PL=0
MOVL C01115 V=800.0 PL=0
MOVL C01116 V=800.0 PL=0
MOVL C01117 V=800.0 PL=0
MOVL C01118 V=800.0 PL=0
MOVL C01119 V=800.0 PL=0
MOVL C01120 V=800.0 PL=0
MOVL C01121 V=800.0 PL=0
MOVL C01122 V=800.0 PL=0
MOVL C01123 V=800.0 PL=0
MOVL C01124 V=800.0 PL=0
MOVL C01125 V=800.0 PL=0
MOVL C01126 V=800.0 PL=0
MOVL C01127 V=800.0 PL=0
MOVL C01128 V=800.0 PL=0
MOVL C01129 V=800.0 PL=0
MOVL C01130 V=800.0 PL=0
MOVL C01131 V=800.0 PL=0
MOVL C01132 V=800.0 PL=0
MOVL C01133 V=800.0 PL=0
MOVL C01134 V=800.0 PL=0
MOVL C01135 V=800.0 PL=0
MOVL C01136 V=800.0 PL=0
MOVL C01137 V=800.0 PL=0
MOVL C01138 V=800.0 PL=0
MOVL C01139 V=800.0 PL=0
MOVL C01140 V=800.0 PL=0
MOVL C01141 V=800.0 PL=0
MOVL C01142 V=800.0 PL=0
MOVL C01143 V=800.0 PL=0
MOVL C01144 V=800.0 PL=0
MOVL C01145 V=800.0 PL=0
MOVL C01146 V=800.0 PL=0
MOVL C01147 V=800.0 PL=0
MOVL C01148 V=800.0 PL=0
MOVL C01149 V=800.0 PL=0
MOVL C01150 V=800.0 PL=0
MOVL C01151 V=800.0 PL=0
MOVL C01152 V=800.0 PL=0
MOVL C01153 V=800.0 PL=0
MOVL C01154 V=800.0 PL=0
MOVL C01155 V=800.0 PL=0
MOVL C01156 V=800.0 PL=0
MOVL C01157 V=800.0 PL=0
MOVL C01158 V=800.0 PL=0
MOVL C01159 V=800.0 PL=0
MOVL C01160 V=800.0 PL=0
MOVL C01161 V=800.0 PL=0
MOVL C01162 V=800.0 PL=0
MOVL C01163 V=800.0 PL=0
MOVL C01164 V=800.0 PL=0
MOVL C01165 V=800.0 PL=0
MOVL C01166 V=800.0 PL=0
MOVL C01167 V=800.0 PL=0
MOVL C01168 V=800.0 PL=0
MOVL C01169 V=800.0 PL=0
MOVL C01170 V=800.0 PL=0
MOVL C01171 V=800.0 PL=0
MOVL C01172 V=800.0 PL=0
MOVL C01173 V=800.0 PL=0
MOVL C01174 V=800.0 PL=0
MOVL C01175 V=800.0 PL=0
MOVL C01176 V=800.0 PL=0
MOVL C01177 V=800.0 PL=0
MOVL C01178 V=800.0 PL=0
MOVL C01179 V=800.0 PL=0
MOVL C01180 V=800.0 PL=0
MOVL C01181 V=800.0 PL=0
MOVL C01182 V=800.0 PL=0
MOVL C01183 V=800.0 PL=0
MOVL C01184 V=800.0 PL=0
MOVL C01185 V=800.0 PL=0
MOVL C01186 V=800.0 PL=0
MOVL C01187 V=800.0 PL=0
MOVL C01188 V=800.0 PL=0
MOVL C01189 V=800.0 PL=0
MOVL C01190 V=800.0 PL=0
MOVL C01191 V=800.0 PL=0
MOVL C01192 V=800.0 PL=0
MOVL C01193 V=800.0 PL=0
MOVL C01194 V=800.0 PL=0
MOVL C01195 V=800.0 PL=0
MOVL C01196 V=800.0 PL=0
MOVL C01197 V=800.0 PL=0
MOVL C01198 V=800.0 PL=0
MOVL C01199 V=800.0 PL=0
MOVL C01200 V=800.0 PL=0
MOVL C01201 V=800.0 PL=0
MOVL C01202 V=800.0 PL=0
MOVL C01203 V=800.0 PL=0
MOVL C01204 V=800.0 PL=0
MOVL C01205 V=800.0 PL=0
MOVL C01206 V=800.0 PL=0
MOVL C01207 V=800.0 PL=0
MOVL C01208 V=800.0 PL=0
MOVL C01209 V=800.0 PL=0
MOVL C01210 V=800.0 PL=0
MOVL C01211 V=800.0 PL=0
MOVL C01212 V=800.0 PL=0
MOVL C01213 V=800.0 PL=0
MOVL C01214 V=800.0 PL=0
MOVL C01215 V=800.0 PL=0
MOVL C01216 V=800.0 PL=0
MOVL C01217 V=800.0 PL=0
MOVL C01218 V=800.0 PL=0
MOVL C01219 V=800.0 PL=0
MOVL C01220 V=800.0 PL=0
MOVL C01221 V=800.0 PL=0
MOVL C01222 V=800.0 PL=0
MOVL C01223 V=800.0 PL=0
MOVL C01224 V=800.0 PL=0
MOVL C01225 V=800.0 PL=0
MOVL C01226 V=800.0 PL=0
MOVL C01227 V=800.0 PL=0
MOVL C01228 V=800.0 PL=0
MOVL C01229 V=800.0 PL=0
MOVL C01230 V=800.0 PL=0
MOVL C01231 V=800.0 PL=0
MOVL C01232 V=800.0 PL=0
MOVL C01233 V=800.0 PL=0
MOVL C01234 V=800.0 PL=0
MOVL C01235 V=800.0 PL=0
MOVL C01236 V=800.0 PL=0
MOVL C01237 V=800.0 PL=0
MOVL C01238 V=800.0 PL=0
MOVL C01239 V=800.0 PL=0
MOVL C01240 V=800.0 PL=0
MOVL C01241 V=800.0 PL=0
MOVL C01242 V=800.0 PL=0
MOVL C01243 V=800.0 PL=0
MOVL C01244 V=800.0 PL=0
MOVL C01245 V=800.0 PL=0
MOVL C01246 V=800.0 PL=0
MOVL C01247 V=800.0 PL=0
MOVL C01248 V=800.0 PL=0
MOVL C01249 V=800.0 PL=0
MOVL C01250 V=800.0 PL=0
MOVL C01251 V=800.0 PL=0
MOVL C01252 V=800.0 PL=0
MOVL C01253 V=800.0 PL=0
MOVL C01254 V=800.0 PL=0
MOVL C01255 V=800.0 PL=0
MOVL C01256 V=800.0 PL=0
MOVL C01257 V=800.0 PL=0
MOVL C01258 V=800.0 PL=0
MOVL C01259 V=800.0 PL=0
MOVL C01260 V=800.0 PL=0
MOVL C01261 V=800.0 PL=0
MOVL C01262 V=800.0 PL=0
MOVL C01263 V=800.0 PL=0
MOVL C01264 V=800.0 PL=0
MOVL C01265 V=800.0 PL=0
MOVL C01266 V=800.0 PL=0
MOVL C01267 V=800.0 PL=0
MOVL C01268 V=800.0 PL=0
MOVL C01269 V=800.0 PL=0
MOVL C01270 V=800.0 PL=0
MOVL C01271 V=800.0 PL=0
MOVL C01272 V=800.0 PL=0
MOVL C01273 V=800.0 PL=0
MOVL C01274 V=800.0 PL=0
MOVL C01275 V=800.0 PL=0
MOVL C01276 V=800.0 PL=0
MOVL C01277 V=800.0 PL=0
MOVL C01278 V=800.0 PL=0
MOVL C01279 V=800.0 PL=0
MOVL C01280 V=800.0 PL=0
MOVL C01281 V=800.0 PL=0
MOVL C01282 V=800.0 PL=0
MOVL C01283 V=800.0 PL=0
MOVL C01284 V=800.0 PL=0
MOVL C01285 V=800.0 PL=0
MOVL C01286 V=800.0 PL=0
MOVL C01287 V=800.0 PL=0
MOVL C01288 V=800.0 PL=0
MOVL C01289 V=800.0 PL=0
MOVL C01290 V=800.0 PL=0
MOVL C01291 V=800.0 PL=0
MOVL C01292 V=800.0 PL=0
MOVL C01293 V=800.0 PL=0
MOVL C01294 V=800.0 PL=0
MOVL C01295 V=800.0 PL=0
MOVL C01296 V=800.0 PL=0
MOVL C01297 V=800.0 PL=0
MOVL C01298 V=800.0 PL=0
MOVL C01299 V=800.0 PL=0
MOVL C01300 V=800.0 PL=0
MOVL C01301 V=800.0 PL=0
MOVL C01302 V=800.0 PL=0
MOVL C01303 V=800.0 PL=0
MOVL C01304 V=800.0 PL=0
MOVL C01305 V=800.0 PL=0
MOVL C01306 V=800.0 PL=0
MOVL C01307 V=800.0 PL=0
MOVL C01308 V=800.0 PL=0
MOVL C01309 V=800.0 PL=0
MOVL C01310 V=800.0 PL=0
MOVL C01311 V=800.0 PL=0
MOVL C01312 V=800.0 PL=0
MOVL C01313 V=800.0 PL=0
MOVL C01314 V=800.0 PL=0
MOVL C01315 V=800.0 PL=0
MOVL C01316 V=800.0 PL=0
MOVL C01317 V=800.0 PL=0
MOVL C01318 V=800.0 PL=0
MOVL C01319 V=800.0 PL=0
MOVL C01320 V=800.0 PL=0
MOVL C01321 V=800.0 PL=0
MOVL C01322 V=800.0 PL=0
MOVL C01323 V=800.0 PL=0
MOVL C01324 V=800.0 PL=0
MOVL C01325 V=800.0 PL=0
MOVL C01326 V=800.0 PL=0
MOVL C01327 V=800.0 PL=0
MOVL C01328 V=800.0 PL=0
MOVL C01329 V=800.0 PL=0
MOVL C01330 V=800.0 PL=0
MOVL C01331 V=800.0 PL=0
MOVL C01332 V=800.0 PL=0
MOVL C01333 V=800.0 PL=0
MOVL C01334 V=800.0 PL=0
MOVL C01335 V=800.0 PL=0
MOVL C01336 V=800.0 PL=0
MOVL C01337 V=800.0 PL=0
MOVL C01338 V=800.0 PL=0
MOVL C01339 V=800.0 PL=0
MOVL C01340 V=800.0 PL=0
MOVL C01341 V=800.0 PL=0
MOVL C01342 V=800.0 PL=0
MOVL C01343 V=800.0 PL=0
MOVL C01344 V=800.0 PL=0
MOVL C01345 V=800.0 PL=0
MOVL C01346 V=800.0 PL=0
MOVL C01347 V=800.0 PL=0
MOVL C01348 V=800.0 PL=0
MOVL C01349 V=800.0 PL=0
MOVL C01350 V=800.0 PL=0
MOVL C01351 V=800.0 PL=0
MOVL C01352 V=800.0 PL=0
MOVL C01353 V=800.0 PL=0
MOVL C01354 V=800.0 PL=0
MOVL C01355 V=800.0 PL=0
MOVL C01356 V=800.0 PL=0
MOVL C01357 V=800.0 PL=0
MOVL C01358 V=800.0 PL=0
MOVL C01359 V=800.0 PL=0
MOVL C01360 V=800.0 PL=0
MOVL C01361 V=800.0 PL=0
MOVL C01362 V=800.0 PL=0
MOVL C01363 V=800.0 PL=0
MOVL C01364 V=800.0 PL=0
MOVL C01365 V=800.0 PL=0
MOVL C01366 V=800.0 PL=0
MOVL C01367 V=800.0 PL=0
MOVL C01368 V=800.0 PL=0
MOVL C01369 V=800.0 PL=0
MOVL C01370 V=800.0 PL=0
MOVL C01371 V=800.0 PL=0
MOVL C01372 V=800.0 PL=0
MOVL C01373 V=800.0 PL=0
MOVL C01374 V=800.0 PL=0
MOVL C01375 V=800.0 PL=0
MOVL C01376 V=800.0 PL=0
MOVL C01377 V=800.0 PL=0
MOVL C01378 V=800.0 PL=0
MOVL C01379 V=800.0 PL=0
MOVL C01380 V=800.0 PL=0
MOVL C01381 V=800.0 PL=0
MOVL C01382 V=800.0 PL=0
MOVL C01383 V=800.0 PL=0
MOVL C01384 V=800.0 PL=0
MOVL C01385 V=800.0 PL=0
MOVL C01386 V=800.0 PL=0
MOVL C01387 V=800.0 PL=0
MOVL C01388 V=800.0 PL=0
MOVL C01389 V=800.0 PL=0
MOVL C01390 V=800.0 PL=0
MOVL C01391 V=800.0 PL=0
MOVL C01392 V=800.0 PL=0
MOVL C01393 V=800.0 PL=0
MOVL C01394 V=800.0 PL=0
MOVL C01395 V=800.0 PL=0
MOVL C01396 V=800.0 PL=0
MOVL C01397 V=800.0 PL=0
MOVL C01398 V=800.0 PL=0
MOVL C01399 V=800.0 PL=0
MOVL C01400 V=800.0 PL=0
MOVL C01401 V=800.0 PL=0
MOVL C01402 V=800.0 PL=0
MOVL C01403 V=800.0 PL=0
MOVL C01404 V=800.0 PL=0
MOVL C01405 V=800.0 PL=0
MOVL C01406 V=800.0 PL=0
MOVL C01407 V=800.0 PL=0
MOVL C01408 V=800.0 PL=0
MOVL C01409 V=800.0 PL=0
MOVL C01410 V=800.0 PL=0
MOVL C01411 V=800.0 PL=0
MOVL C01412 V=800.0 PL=0
MOVL C01413 V=800.0 PL=0
MOVL C01414 V=800.0 PL=0
MOVL C01415 V=800.0 PL=0
MOVL C01416 V=800.0 PL=0
MOVL C01417 V=800.0 PL=0
MOVL C01418 V=800.0 PL=0
MOVL C01419 V=800.0 PL=0
MOVL C01420 V=800.0 PL=0
MOVL C01421 V=800.0 PL=0
MOVL C01422 V=800.0 PL=0
MOVL C01423 V=800.0 PL=0
MOVL C01424 V=800.0 PL=0
MOVL C01425 V=800.0 PL=0
MOVL C01426 V=800.0 PL=0
MOVL C01427 V=800.0 PL=0
MOVL C01428 V=800.0 PL=0
MOVL C01429 V=800.0 PL=0
MOVL C01430 V=800.0 PL=0
MOVL C01431 V=800.0 PL=0
MOVL C01432 V=800.0 PL=0
MOVL C01433 V=800.0 PL=0
MOVL C01434 V=800.0 PL=0
MOVL C01435 V=800.0 PL=0
MOVL C01436 V=800.0 PL=0
MOVL C01437 V=800.0 PL=0
MOVL C01438 V=800.0 PL=0
MOVL C01439 V=800.0 PL=0
MOVL C01440 V=800.0 PL=0
MOVL C01441 V=800.0 PL=0
MOVL C01442 V=800.0 PL=0
MOVL C01443 V=800.0 PL=0
MOVL C01444 V=800.0 PL=0
MOVL C01445 V=800.0 PL=0
MOVL C01446 V=800.0 PL=0
MOVL C01447 V=800.0 PL=0
MOVL C01448 V=800.0 PL=0
MOVL C01449 V=800.0 PL=0
MOVL C01450 V=800.0 PL=0
MOVL C01451 V=800.0 PL=0
MOVL C01452 V=800.0 PL=0
MOVL C01453 V=800.0 PL=0
MOVL C01454 V=800.0 PL=0
MOVL C01455 V=800.0 PL=0
MOVL C01456 V=800.0 PL=0
MOVL C01457 V=800.0 PL=0
MOVL C01458 V=800.0 PL=0
MOVL C01459 V=800.0 PL=0
MOVL C01460 V=800.0 PL=0
MOVL C01461 V=800.0 PL=0
MOVL C01462 V=800.0 PL=0
MOVL C01463 V=800.0 PL=0
MOVL C01464 V=800.0 PL=0
MOVL C01465 V=800.0 PL=0
MOVL C01466 V=800.0 PL=0
MOVL C01467 V=800.0 PL=0
MOVL C01468 V=800.0 PL=0
MOVL C01469 V=800.0 PL=0
MOVL C01470 V=800.0 PL=0
MOVL C01471 V=800.0 PL=0
MOVL C01472 V=800.0 PL=0
MOVL C01473 V=800.0 PL=0
MOVL C01474 V=800.0 PL=0
MOVL C01475 V=800.0 PL=0
MOVL C01476 V=800.0 PL=0
MOVL C01477 V=800.0 PL=0
MOVL C01478 V=800.0 PL=0
MOVL C01479 V=800.0 PL=0
MOVL C01480 V=800.0 PL=0
MOVL C01481 V=800.0 PL=0
MOVL C01482 V=800.0 PL=0
MOVL C01483 V=800.0 PL=0
MOVL C01484 V=800.0 PL=0
MOVL C01485 V=800.0 PL=0
MOVL C01486 V=800.0 PL=0
MOVL C01487 V=800.0 PL=0
MOVL C01488 V=800.0 PL=0
MOVL C01489 V=800.0 PL=0
MOVL C01490 V=800.0 PL=0
MOVL C01491 V=800.0 PL=0
MOVL C01492 V=800.0 PL=0
MOVL C01493 V=800.0 PL=0
MOVL C01494 V=800.0 PL=0
MOVL C01495 V=800.0 PL=0
MOVL C01496 V=800.0 PL=0
MOVL C01497 V=800.0 PL=0
MOVL C01498 V=800.0 PL=0
MOVL C01499 V=800.0 PL=0
MOVL C01500 V=800.0 PL=0
MOVL C01501 V=800.0 PL=0
MOVL C01502 V=800.0 PL=0
MOVL C01503 V=800.0 PL=0
MOVL C01504 V=800.0 PL=0
MOVL C01505 V=800.0 PL=0
MOVL C01506 V=800.0 PL=0
MOVL C01507 V=800.0 PL=0
MOVL C01508 V=800.0 PL=0
MOVL C01509 V=800.0 PL=0
MOVL C01510 V=800.0 PL=0
MOVL C01511 V=800.0 PL=0
MOVL C01512 V=800.0 PL=0
MOVL C01513 V=800.0 PL=0
MOVL C01514 V=800.0 PL=0
MOVL C01515 V=800.0 PL=0
MOVL C01516 V=800.0 PL=0
MOVL C01517 V=800.0 PL=0
MOVL C01518 V=800.0 PL=0
MOVL C01519 V=800.0 PL=0
MOVL C01520 V=800.0 PL=0
MOVL C01521 V=800.0 PL=0
MOVL C01522 V=800.0 PL=0
MOVL C01523 V=800.0 PL=0
MOVL C01524 V=800.0 PL=0
MOVL C01525 V=800.0 PL=0
MOVL C01526 V=800.0 PL=0
MOVL C01527 V=800.0 PL=0
MOVL C01528 V=800.0 PL=0
MOVL C01529 V=800.0 PL=0
MOVL C01530 V=800.0 PL=0
MOVL C01531 V=800.0 PL=0
MOVL C01532 V=800.0 PL=0
MOVL C01533 V=800.0 PL=0
MOVL C01534 V=800.0 PL=0
MOVL C01535 V=800.0 PL=0
MOVL C01536 V=800.0 PL=0
MOVL C01537 V=800.0 PL=0
MOVL C01538 V=800.0 PL=0
MOVL C01539 V=800.0 PL=0
MOVL C01540 V=800.0 PL=0
MOVL C01541 V=800.0 PL=0
MOVL C01542 V=800.0 PL=0
MOVL C01543 V=800.0 PL=0
MOVL C01544 V=800.0 PL=0
MOVL C01545 V=800.0 PL=0
MOVL C01546 V=800.0 PL=0
MOVL C01547 V=800.0 PL=0
MOVL C01548 V=800.0 PL=0
MOVL C01549 V=800.0 PL=0
MOVL C01550 V=800.0 PL=0
MOVL C01551 V=800.0 PL=0
MOVL C01552 V=800.0 PL=0
MOVL C01553 V=800.0 PL=0
MOVL C01554 V=800.0 PL=0
MOVL C01555 V=800.0 PL=0
MOVL C01556 V=800.0 PL=0
MOVL C01557 V=800.0 PL=0
MOVL C01558 V=800.0 PL=0
MOVL C01559 V=800.0 PL=0
MOVL C01560 V=800.0 PL=0
MOVL C01561 V=800.0 PL=0
MOVL C01562 V=800.0 PL=0
MOVL C01563 V=800.0 PL=0
MOVL C01564 V=800.0 PL=0
MOVL C01565 V=800.0 PL=0
MOVL C01566 V=800.0 PL=0
MOVL C01567 V=800.0 PL=0
MOVL C01568 V=800.0 PL=0
MOVL C01569 V=800.0 PL=0
MOVL C01570 V=800.0 PL=0
MOVL C01571 V=800.0 PL=0
MOVL C01572 V=800.0 PL=0
MOVL C01573 V=800.0 PL=0
MOVL C01574 V=800.0 PL=0
MOVL C01575 V=800.0 PL=0
MOVL C01576 V=800.0 PL=0
MOVL C01577 V=800.0 PL=0
MOVL C01578 V=800.0 PL=0
MOVL C01579 V=800.0 PL=0
MOVL C01580 V=800.0 PL=0
MOVL C01581 V=800.0 PL=0
MOVL C01582 V=800.0 PL=0
MOVL C01583 V=800.0 PL=0
MOVL C01584 V=800.0 PL=0
MOVL C01585 V=800.0 PL=0
MOVL C01586 V=800.0 PL=0
MOVL C01587 V=800.0 PL=0
MOVL C01588 V=800.0 PL=0
MOVL C01589 V=800.0 PL=0
MOVL C01590 V=800.0 PL=0
MOVL C01591 V=800.0 PL=0
MOVL C01592 V=800.0 PL=0
MOVL C01593 V=800.0 PL=0
MOVL C01594 V=800.0 PL=0
MOVL C01595 V=800.0 PL=0
MOVL C01596 V=800.0 PL=0
MOVL C01597 V=800.0 PL=0
MOVL C01598 V=800.0 PL=0
MOVL C01599 V=800.0 PL=0
MOVL C01600 V=800.0 PL=0
MOVL C01601 V=800.0 PL=0
MOVL C01602 V=800.0 PL=0
MOVL C01603 V=800.0 PL=0
MOVL C01604 V=800.0 PL=0
MOVL C01605 V=800.0 PL=0
MOVL C01606 V=800.0 PL=0
MOVL C01607 V=800.0 PL=0
MOVL C01608 V=800.0 PL=0
MOVL C01609 V=800.0 PL=0
MOVL C01610 V=800.0 PL=0
MOVL C01611 V=800.0 PL=0
MOVL C01612 V=800.0 PL=0
MOVL C01613 V=800.0 PL=0
MOVL C01614 V=800.0 PL=0
MOVL C01615 V=800.0 PL=0
MOVL C01616 V=800.0 PL=0
MOVL C01617 V=800.0 PL=0
MOVL C01618 V=800.0 PL=0
MOVL C01619 V=800.0 PL=0
MOVL C01620 V=800.0 PL=0
MOVL C01621 V=800.0 PL=0
MOVL C01622 V=800.0 PL=0
MOVL C01623 V=800.0 PL=0
MOVL C01624 V=800.0 PL=0
MOVL C01625 V=800.0 PL=0
MOVL C01626 V=800.0 PL=0
MOVL C01627 V=800.0 PL=0
MOVL C01628 V=800.0 PL=0
MOVL C01629 V=800.0 PL=0
MOVL C01630 V=800.0 PL=0
MOVL C01631 V=800.0 PL=0
MOVL C01632 V=800.0 PL=0
MOVL C01633 V=800.0 PL=0
MOVL C01634 V=800.0 PL=0
MOVL C01635 V=800.0 PL=0
MOVL C01636 V=800.0 PL=0
MOVL C01637 V=800.0 PL=0
MOVL C01638 V=800.0 PL=0
MOVL C01639 V=800.0 PL=0
MOVL C01640 V=800.0 PL=0
MOVL C01641 V=800.0 PL=0
MOVL C01642 V=800.0 PL=0
MOVL C01643 V=800.0 PL=0
MOVL C01644 V=800.0 PL=0
MOVL C01645 V=800.0 PL=0
MOVL C01646 V=800.0 PL=0
MOVL C01647 V=800.0 PL=0
MOVL C01648 V=800.0 PL=0
MOVL C01649 V=800.0 PL=0
MOVL C01650 V=800.0 PL=0
MOVL C01651 V=800.0 PL=0
MOVL C01652 V=800.0 PL=0
MOVL C01653 V=800.0 PL=0
MOVL C01654 V=800.0 PL=0
MOVL C01655 V=800.0 PL=0
MOVL C01656 V=800.0 PL=0
MOVL C01657 V=800.0 PL=0
MOVL C01658 V=800.0 PL=0
MOVL C01659 V=800.0 PL=0
MOVL C01660 V=800.0 PL=0
MOVL C01661 V=800.0 PL=0
MOVL C01662 V=800.0 PL=0
MOVL C01663 V=800.0 PL=0
MOVL C01664 V=800.0 PL=0
MOVL C01665 V=800.0 PL=0
MOVL C01666 V=800.0 PL=0
MOVL C01667 V=800.0 PL=0
MOVL C01668 V=800.0 PL=0
MOVL C01669 V=800.0 PL=0
MOVL C01670 V=800.0 PL=0
MOVL C01671 V=800.0 PL=0
MOVL C01672 V=800.0 PL=0
MOVL C01673 V=800.0 PL=0
MOVL C01674 V=800.0 PL=0
MOVL C01675 V=800.0 PL=0
MOVL C01676 V=800.0 PL=0
MOVL C01677 V=800.0 PL=0
MOVL C01678 V=800.0 PL=0
MOVL C01679 V=800.0 PL=0
MOVL C01680 V=800.0 PL=0
MOVL C01681 V=800.0 PL=0
MOVL C01682 V=800.0 PL=0
MOVL C01683 V=800.0 PL=0
MOVL C01684 V=800.0 PL=0
MOVL C01685 V=800.0 PL=0
MOVL C01686 V=800.0 PL=0
MOVL C01687 V=800.0 PL=0
MOVL C01688 V=800.0 PL=0
MOVL C01689 V=800.0 PL=0
MOVL C01690 V=800.0 PL=0
MOVL C01691 V=800.0 PL=0
MOVL C01692 V=800.0 PL=0
MOVL C01693 V=800.0 PL=0
MOVL C01694 V=800.0 PL=0
MOVL C01695 V=800.0 PL=0
MOVL C01696 V=800.0 PL=0
MOVL C01697 V=800.0 PL=0
MOVL C01698 V=800.0 PL=0
MOVL C01699 V=800.0 PL=0
MOVL C01700 V=800.0 PL=0
MOVL C01701 V=800.0 PL=0
MOVL C01702 V=800.0 PL=0
MOVL C01703 V=800.0 PL=0
MOVL C01704 V=800.0 PL=0
MOVL C01705 V=800.0 PL=0
MOVL C01706 V=800.0 PL=0
MOVL C01707 V=800.0 PL=0
MOVL C01708 V=800.0 PL=0
MOVL C01709 V=800.0 PL=0
MOVL C01710 V=800.0 PL=0
MOVL C01711 V=800.0 PL=0
MOVL C01712 V=800.0 PL=0
MOVL C01713 V=800.0 PL=0
MOVL C01714 V=800.0 PL=0
MOVL C01715 V=800.0 PL=0
MOVL C01716 V=800.0 PL=0
MOVL C01717 V=800.0 PL=0
MOVL C01718 V=800.0 PL=0
MOVL C01719 V=800.0 PL=0
MOVL C01720 V=800.0 PL=0
MOVL C01721 V=800.0 PL=0
MOVL C01722 V=800.0 PL=0
MOVL C01723 V=800.0 PL=0
MOVL C01724 V=800.0 PL=0
MOVL C01725 V=800.0 PL=0
MOVL C01726 V=800.0 PL=0
MOVL C01727 V=800.0 PL=0
MOVL C01728 V=800.0 PL=0
MOVL C01729 V=800.0 PL=0
MOVL C01730 V=800.0 PL=0
MOVL C01731 V=800.0 PL=0
MOVL C01732 V=800.0 PL=0
MOVL C01733 V=800.0 PL=0
MOVL C01734 V=800.0 PL=0
MOVL C01735 V=800.0 PL=0
MOVL C01736 V=800.0 PL=0
MOVL C01737 V=800.0 PL=0
MOVL C01738 V=800.0 PL=0
MOVL C01739 V=800.0 PL=0
MOVL C01740 V=800.0 PL=0
MOVL C01741 V=800.0 PL=0
MOVL C01742 V=800.0 PL=0
MOVL C01743 V=800.0 PL=0
MOVL C01744 V=800.0 PL=0
MOVL C01745 V=800.0 PL=0
MOVL C01746 V=800.0 PL=0
MOVL C01747 V=800.0 PL=0
MOVL C01748 V=800.0 PL=0
MOVL C01749 V=800.0 PL=0
MOVL C01750 V=800.0 PL=0
MOVL C01751 V=800.0 PL=0
MOVL C01752 V=800.0 PL=0
MOVL C01753 V=800.0 PL=0
MOVL C01754 V=800.0 PL=0
MOVL C01755 V=800.0 PL=0
MOVL C01756 V=800.0 PL=0
MOVL C01757 V=800.0 PL=0
MOVL C01758 V=800.0 PL=0
MOVL C01759 V=800.0 PL=0
MOVL C01760 V=800.0 PL=0
MOVL C01761 V=800.0 PL=0
MOVL C01762 V=800.0 PL=0
MOVL C01763 V=800.0 PL=0
MOVL C01764 V=800.0 PL=0
MOVL C01765 V=800.0 PL=0
MOVL C01766 V=800.0 PL=0
MOVL C01767 V=800.0 PL=0
MOVL C01768 V=800.0 PL=0
MOVL C01769 V=800.0 PL=0
MOVL C01770 V=800.0 PL=0
MOVL C01771 V=800.0 PL=0
MOVL C01772 V=800.0 PL=0
MOVL C01773 V=800.0 PL=0
MOVL C01774 V=800.0 PL=0
MOVL C01775 V=800.0 PL=0
MOVL C01776 V=800.0 PL=0
MOVL C01777 V=800.0 PL=0
MOVL C01778 V=800.0 PL=0
MOVL C01779 V=800.0 PL=0
MOVL C01780 V=800.0 PL=0
MOVL C01781 V=800.0 PL=0
MOVL C01782 V=800.0 PL=0
MOVL C01783 V=800.0 PL=0
MOVL C01784 V=800.0 PL=0
MOVL C01785 V=800.0 PL=0
MOVL C01786 V=800.0 PL=0
MOVL C01787 V=800.0 PL=0
MOVL C01788 V=800.0 PL=0
MOVL C01789 V=800.0 PL=0
MOVL C01790 V=800.0 PL=0
MOVL C01791 V=800.0 PL=0
MOVL C01792 V=800.0 PL=0
MOVL C01793 V=800.0 PL=0
MOVL C01794 V=800.0 PL=0
MOVL C01795 V=800.0 PL=0
MOVL C01796 V=800.0 PL=0
MOVL C01797 V=800.0 PL=0
MOVL C01798 V=800.0 PL=0
MOVL C01799 V=800.0 PL=0
MOVL C01800 V=800.0 PL=0
MOVL C01801 V=800.0 PL=0
MOVL C01802 V=800.0 PL=0
MOVL C01803 V=800.0 PL=0
MOVL C01804 V=800.0 PL=0
MOVL C01805 V=800.0 PL=0
MOVL C01806 V=800.0 PL=0
MOVL C01807 V=800.0 PL=0
MOVL C01808 V=800.0 PL=0
MOVL C01809 V=800.0 PL=0
MOVL C01810 V=800.0 PL=0
MOVL C01811 V=800.0 PL=0
MOVL C01812 V=800.0 PL=0
MOVL C01813 V=800.0 PL=0
MOVL C01814 V=800.0 PL=0
MOVL C01815 V=800.0 PL=0
MOVL C01816 V=800.0 PL=0
MOVL C01817 V=800.0 PL=0
MOVL C01818 V=800.0 PL=0
MOVL C01819 V=800.0 PL=0
MOVL C01820 V=800.0 PL=0
MOVL C01821 V=800.0 PL=0
MOVL C01822 V=800.0 PL=0
MOVL C01823 V=800.0 PL=0
MOVL C01824 V=800.0 PL=0
MOVL C01825 V=800.0 PL=0
MOVL C01826 V=800.0 PL=0
MOVL C01827 V=800.0 PL=0
MOVL C01828 V=800.0 PL=0
MOVL C01829 V=800.0 PL=0
MOVL C01830 V=800.0 PL=0
MOVL C01831 V=800.0 PL=0
MOVL C01832 V=800.0 PL=0
MOVL C01833 V=800.0 PL=0
MOVL C01834 V=800.0 PL=0
MOVL C01835 V=800.0 PL=0
MOVL C01836 V=800.0 PL=0
MOVL C01837 V=800.0 PL=0
MOVL C01838 V=800.0 PL=0
MOVL C01839 V=800.0 PL=0
MOVL C01840 V=800.0 PL=0
MOVL C01841 V=800.0 PL=0
MOVL C01842 V=800.0 PL=0
MOVL C01843 V=800.0 PL=0
MOVL C01844 V=800.0 PL=0
MOVL C01845 V=800.0 PL=0
MOVL C01846 V=800.0 PL=0
MOVL C01847 V=800.0 PL=0
MOVL C01848 V=800.0 PL=0
MOVL C01849 V=800.0 PL=0
MOVL C01850 V=800.0 PL=0
MOVL C01851 V=800.0 PL=0
MOVL C01852 V=800.0 PL=0
MOVL C01853 V=800.0 PL=0
MOVL C01854 V=800.0 PL=0
MOVL C01855 V=800.0 PL=0
MOVL C01856 V=800.0 PL=0
MOVL C01857 V=800.0 PL=0
MOVL C01858 V=800.0 PL=0
MOVL C01859 V=800.0 PL=0
MOVL C01860 V=800.0 PL=0
MOVL C01861 V=800.0 PL=0
MOVL C01862 V=800.0 PL=0
MOVL C01863 V=800.0 PL=0
MOVL C01864 V=800.0 PL=0
MOVL C01865 V=800.0 PL=0
MOVL C01866 V=800.0 PL=0
MOVL C01867 V=800.0 PL=0
MOVL C01868 V=800.0 PL=0
MOVL C01869 V=800.0 PL=0
MOVL C01870 V=800.0 PL=0
MOVL C01871 V=800.0 PL=0
MOVL C01872 V=800.0 PL=0
MOVL C01873 V=800.0 PL=0
MOVL C01874 V=800.0 PL=0
MOVL C01875 V=800.0 PL=0
MOVL C01876 V=800.0 PL=0
MOVL C01877 V=800.0 PL=0
MOVL C01878 V=800.0 PL=0
MOVL C01879 V=800.0 PL=0
MOVL C01880 V=800.0 PL=0
MOVL C01881 V=800.0 PL=0
MOVL C01882 V=800.0 PL=0
MOVL C01883 V=800.0 PL=0
MOVL C01884 V=800.0 PL=0
MOVL C01885 V=800.0 PL=0
MOVL C01886 V=800.0 PL=0
MOVL C01887 V=800.0 PL=0
MOVL C01888 V=800.0 PL=0
MOVL C01889 V=800.0 PL=0
MOVL C01890 V=800.0 PL=0
MOVL C01891 V=800.0 PL=0
MOVL C01892 V=800.0 PL=0
MOVL C01893 V=800.0 PL=0
MOVL C01894 V=800.0 PL=0
MOVL C01895 V=800.0 PL=0
MOVL C01896 V=800.0 PL=0
MOVL C01897 V=800.0 PL=0
MOVL C01898 V=800.0 PL=0
MOVL C01899 V=800.0 PL=0
MOVL C01900 V=800.0 PL=0
MOVL C01901 V=800.0 PL=0
MOVL C01902 V=800.0 PL=0
MOVL C01903 V=800.0 PL=0
MOVL C01904 V=800.0 PL=0
MOVL C01905 V=800.0 PL=0
MOVL C01906 V=800.0 PL=0
MOVL C01907 V=800.0 PL=0
MOVL C01908 V=800.0 PL=0
MOVL C01909 V=800.0 PL=0
MOVL C01910 V=800.0 PL=0
MOVL C01911 V=800.0 PL=0
MOVL C01912 V=800.0 PL=0
MOVL C01913 V=800.0 PL=0
MOVL C01914 V=800.0 PL=0
MOVL C01915 V=800.0 PL=0
MOVL C01916 V=800.0 PL=0
MOVL C01917 V=800.0 PL=0
MOVL C01918 V=800.0 PL=0
MOVL C01919 V=800.0 PL=0
MOVL C01920 V=800.0 PL=0
MOVL C01921 V=800.0 PL=0
MOVL C01922 V=800.0 PL=0
MOVL C01923 V=800.0 PL=0
MOVL C01924 V=800.0 PL=0
MOVL C01925 V=800.0 PL=0
MOVL C01926 V=800.0 PL=0
MOVL C01927 V=800.0 PL=0
MOVL C01928 V=800.0 PL=0
MOVL C01929 V=800.0 PL=0
MOVL C01930 V=800.0 PL=0
MOVL C01931 V=800.0 PL=0
MOVL C01932 V=800.0 PL=0
MOVL C01933 V=800.0 PL=0
MOVL C01934 V=800.0 PL=0
MOVL C01935 V=800.0 PL=0
MOVL C01936 V=800.0 PL=0
MOVL C01937 V=800.0 PL=0
MOVL C01938 V=800.0 PL=0
MOVL C01939 V=800.0 PL=0
MOVL C01940 V=800.0 PL=0
MOVL C01941 V=800.0 PL=0
MOVL C01942 V=800.0 PL=0
MOVL C01943 V=800.0 PL=0
MOVL C01944 V=800.0 PL=0
MOVL C01945 V=800.0 PL=0
MOVL C01946 V=800.0 PL=0
MOVL C01947 V=800.0 PL=0
MOVL C01948 V=800.0 PL=0
MOVL C01949 V=800.0 PL=0
MOVL C01950 V=800.0 PL=0
MOVL C01951 V=800.0 PL=0
MOVL C01952 V=800.0 PL=0
MOVL C01953 V=800.0 PL=0
MOVL C01954 V=800.0 PL=0
MOVL C01955 V=800.0 PL=0
MOVL C01956 V=800.0 PL=0
MOVL C01957 V=800.0 PL=0
MOVL C01958 V=800.0 PL=0
MOVL C01959 V=800.0 PL=0
MOVL C01960 V=800.0 PL=0
MOVL C01961 V=800.0 PL=0
MOVL C01962 V=800.0 PL=0
MOVL C01963 V=800.0 PL=0
MOVL C01964 V=800.0 PL=0
MOVL C01965 V=800.0 PL=0
MOVL C01966 V=800.0 PL=0
MOVL C01967 V=800.0 PL=0
MOVL C01968 V=800.0 PL=0
MOVL C01969 V=800.0 PL=0
MOVL C01970 V=800.0 PL=0
MOVL C01971 V=800.0 PL=0
MOVL C01972 V=800.0 PL=0
MOVL C01973 V=800.0 PL=0
MOVL C01974 V=800.0 PL=0
MOVL C01975 V=800.0 PL=0
MOVL C01976 V=800.0 PL=0
MOVL C01977 V=800.0 PL=0
MOVL C01978 V=800.0 PL=0
MOVL C01979 V=800.0 PL=0
MOVL C01980 V=800.0 PL=0
MOVL C01981 V=800.0 PL=0
MOVL C01982 V=800.0 PL=0
MOVL C01983 V=800.0 PL=0
MOVL C01984 V=800.0 PL=0
MOVL C01985 V=800.0 PL=0
MOVL C01986 V=800.0 PL=0
MOVL C01987 V=800.0 PL=0
MOVL C01988 V=800.0 PL=0
MOVL C01989 V=800.0 PL=0
MOVL C01990 V=800.0 PL=0
MOVL C01991 V=800.0 PL=0
MOVL C01992 V=800.0 PL=0
MOVL C01993 V=800.0 PL=0
MOVL C01994 V=800.0 PL=0
MOVL C01995 V=800.0 PL=0
MOVL C01996 V=800.0 PL=0
MOVL C01997 V=800.0 PL=0
MOVL C01998 V=800.0 PL=0
MOVL C01999 V=800.0 PL=0
MOVL C02000 V=800.0 PL=0
MOVL C02001 V=800.0 PL=0
MOVL C02002 V=800.0 PL=0
MOVL C02003 V=800.0 PL=0
MOVL C02004 V=800.0 PL=0
MOVL C02005 V=800.0 PL=0
MOVL C02006 V=800.0 PL=0
MOVL C02007 V=800.0 PL=0
MOVL C02008 V=800.0 PL=0
MOVL C02009 V=800.0 PL=0
MOVL C02010 V=800.0 PL=0
MOVL C02011 V=800.0 PL=0
MOVL C02012 V=800.0 PL=0
MOVL C02013 V=800.0 PL=0
MOVL C02014 V=800.0 PL=0
MOVL C02015 V=800.0 PL=0
MOVL C02016 V=800.0 PL=0
MOVL C02017 V=800.0 PL=0
MOVL C02018 V=800.0 PL=0
MOVL C02019 V=800.0 PL=0
MOVL C02020 V=800.0 PL=0
MOVL C02021 V=800.0 PL=0
MOVL C02022 V=800.0 PL=0
MOVL C02023 V=800.0 PL=0
MOVL C02024 V=800.0 PL=0
MOVL C02025 V=800.0 PL=0
MOVL C02026 V=800.0 PL=0
MOVL C02027 V=800.0 PL=0
MOVL C02028 V=800.0 PL=0
MOVL C02029 V=800.0 PL=0
MOVL C02030 V=800.0 PL=0
MOVL C02031 V=800.0 PL=0
MOVL C02032 V=800.0 PL=0
MOVL C02033 V=800.0 PL=0
MOVL C02034 V=800.0 PL=0
MOVL C02035 V=800.0 PL=0
MOVL C02036 V=800.0 PL=0
MOVL C02037 V=800.0 PL=0
MOVL C02038 V=800.0 PL=0
MOVL C02039 V=800.0 PL=0
MOVL C02040 V=800.0 PL=0
MOVL C02041 V=800.0 PL=0
MOVL C02042 V=800.0 PL=0
MOVL C02043 V=800.0 PL=0
MOVL C02044 V=800.0 PL=0
MOVL C02045 V=800.0 PL=0
MOVL C02046 V=800.0 PL=0
MOVL C02047 V=800.0 PL=0
MOVL C02048 V=800.0 PL=0
MOVL C02049 V=800.0 PL=0
MOVL C02050 V=800.0 PL=0
MOVL C02051 V=800.0 PL=0
MOVL C02052 V=800.0 PL=0
MOVL C02053 V=800.0 PL=0
MOVL C02054 V=800.0 PL=0
MOVL C02055 V=800.0 PL=0
MOVL C02056 V=800.0 PL=0
MOVL C02057 V=800.0 PL=0
MOVL C02058 V=800.0 PL=0
MOVL C02059 V=800.0 PL=0
MOVL C02060 V=800.0 PL=0
MOVL C02061 V=800.0 PL=0
MOVL C02062 V=800.0 PL=0
MOVL C02063 V=800.0 PL=0
MOVL C02064 V=800.0 PL=0
MOVL C02065 V=800.0 PL=0
MOVL C02066 V=800.0 PL=0
MOVL C02067 V=800.0 PL=0
MOVL C02068 V=800.0 PL=0
MOVL C02069 V=800.0 PL=0
MOVL C02070 V=800.0 PL=0
MOVL C02071 V=800.0 PL=0
MOVL C02072 V=800.0 PL=0
MOVL C02073 V=800.0 PL=0
MOVL C02074 V=800.0 PL=0
MOVL C02075 V=800.0 PL=0
MOVL C02076 V=800.0 PL=0
MOVL C02077 V=800.0 PL=0
MOVL C02078 V=800.0 PL=0
MOVL C02079 V=800.0 PL=0
MOVL C02080 V=800.0 PL=0
MOVL C02081 V=800.0 PL=0
MOVL C02082 V=800.0 PL=0
MOVL C02083 V=800.0 PL=0
MOVL C02084 V=800.0 PL=0
MOVL C02085 V=800.0 PL=0
MOVL C02086 V=800.0 PL=0
MOVL C02087 V=800.0 PL=0
MOVL C02088 V=800.0 PL=0
MOVL C02089 V=800.0 PL=0
MOVL C02090 V=800.0 PL=0
MOVL C02091 V=800.0 PL=0
MOVL C02092 V=800.0 PL=0
MOVL C02093 V=800.0 PL=0
MOVL C02094 V=800.0 PL=0
MOVL C02095 V=800.0 PL=0
MOVL C02096 V=800.0 PL=0
MOVL C02097 V=800.0 PL=0
MOVL C02098 V=800.0 PL=0
MOVL C02099 V=800.0 PL=0
MOVL C02100 V=800.0 PL=0
MOVL C02101 V=800.0 PL=0
MOVL C02102 V=800.0 PL=0
MOVL C02103 V=800.0 PL=0
MOVL C02104 V=800.0 PL=0
MOVL C02105 V=800.0 PL=0
MOVL C02106 V=800.0 PL=0
MOVL C02107 V=800.0 PL=0
MOVL C02108 V=800.0 PL=0
MOVL C02109 V=800.0 PL=0
MOVL C02110 V=800.0 PL=0
MOVL C02111 V=800.0 PL=0
MOVL C02112 V=800.0 PL=0
MOVL C02113 V=800.0 PL=0
MOVL C02114 V=800.0 PL=0
